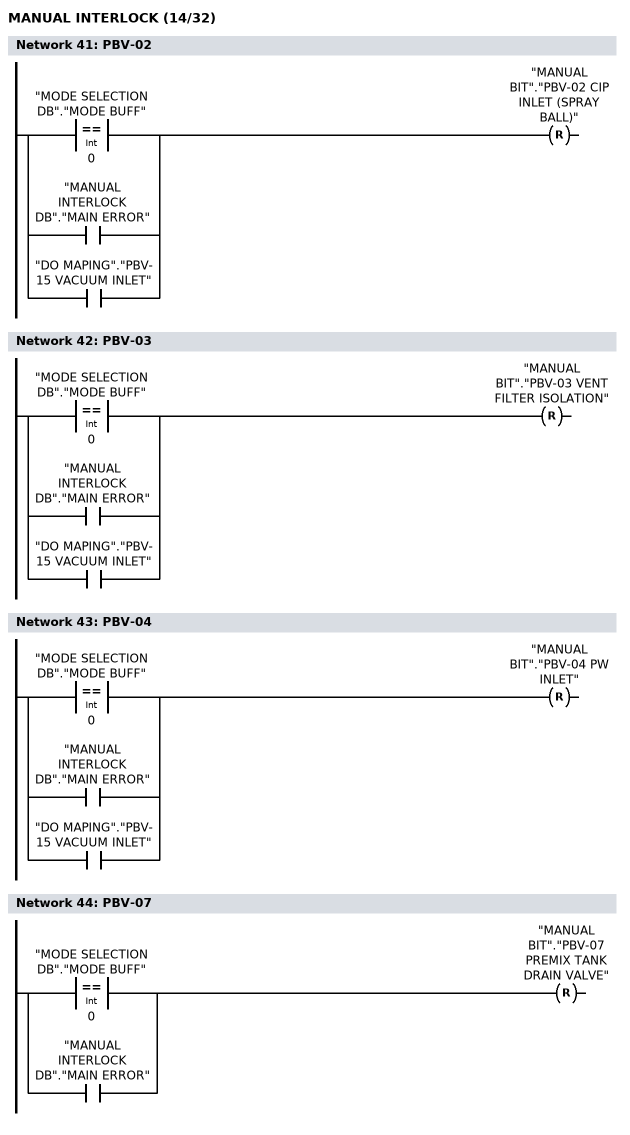
   RUNG wire#powerrail
      { S7_Templates := "SrcType := Int" } EQ_Contact(in1 := "MODE SELECTION DB"."MODE BUFF", in2 := 0)
      wire#w1
      R_Coil( "MANUAL BIT"."PBV-02 CIP INLET (SPRAY BALL)" )
   END_RUNG
   RUNG wire#powerrail
      Contact( "MANUAL INTERLOCK DB"."MAIN ERROR" )
   END_RUNG wire#w1
   RUNG wire#powerrail
      Contact( "DO MAPING"."PBV-15 VACUUM INLET" )
   END_RUNG wire#w1
   // the same network as SCL:
   IF ("MODE SELECTION DB"."MODE BUFF" = 0) OR "MANUAL INTERLOCK DB"."MAIN ERROR" OR "DO MAPING"."PBV-15 VACUUM INLET" THEN
       "MANUAL BIT"."PBV-02 CIP INLET (SPRAY BALL)" := FALSE;
   END_IF;
END_REGION

REGION Network 42: PBV-03
   RUNG wire#powerrail
      { S7_Templates := "SrcType := Int" } EQ_Contact(in1 := "MODE SELECTION DB"."MODE BUFF", in2 := 0)
      wire#w1
      R_Coil( "MANUAL BIT"."PBV-03 VENT FILTER ISOLATION" )
   END_RUNG
   RUNG wire#powerrail
      Contact( "MANUAL INTERLOCK DB"."MAIN ERROR" )
   END_RUNG wire#w1
   RUNG wire#powerrail
      Contact( "DO MAPING"."PBV-15 VACUUM INLET" )
   END_RUNG wire#w1
   // the same network as SCL:
   IF ("MODE SELECTION DB"."MODE BUFF" = 0) OR "MANUAL INTERLOCK DB"."MAIN ERROR" OR "DO MAPING"."PBV-15 VACUUM INLET" THEN
       "MANUAL BIT"."PBV-03 VENT FILTER ISOLATION" := FALSE;
   END_IF;
END_REGION

REGION Network 43: PBV-04
   RUNG wire#powerrail
      { S7_Templates := "SrcType := Int" } EQ_Contact(in1 := "MODE SELECTION DB"."MODE BUFF", in2 := 0)
      wire#w1
      R_Coil( "MANUAL BIT"."PBV-04 PW INLET" )
   END_RUNG
   RUNG wire#powerrail
      Contact( "MANUAL INTERLOCK DB"."MAIN ERROR" )
   END_RUNG wire#w1
   RUNG wire#powerrail
      Contact( "DO MAPING"."PBV-15 VACUUM INLET" )
   END_RUNG wire#w1
   // the same network as SCL:
   IF ("MODE SELECTION DB"."MODE BUFF" = 0) OR "MANUAL INTERLOCK DB"."MAIN ERROR" OR "DO MAPING"."PBV-15 VACUUM INLET" THEN
       "MANUAL BIT"."PBV-04 PW INLET" := FALSE;
   END_IF;
END_REGION

REGION Network 44: PBV-07
   RUNG wire#powerrail
      { S7_Templates := "SrcType := Int" } EQ_Contact(in1 := "MODE SELECTION DB"."MODE BUFF", in2 := 0)
      wire#w1
      R_Coil( "MANUAL BIT"."PBV-07 PREMIX TANK DRAIN VALVE" )
   END_RUNG
   RUNG wire#powerrail
      Contact( "MANUAL INTERLOCK DB"."MAIN ERROR" )
   END_RUNG wire#w1
   // the same network as SCL:
   IF ("MODE SELECTION DB"."MODE BUFF" = 0) OR "MANUAL INTERLOCK DB"."MAIN ERROR" THEN
       "MANUAL BIT"."PBV-07 PREMIX TANK DRAIN VALVE" := FALSE;
   END_IF;
END_REGION

REGION Network 45: PAV-09
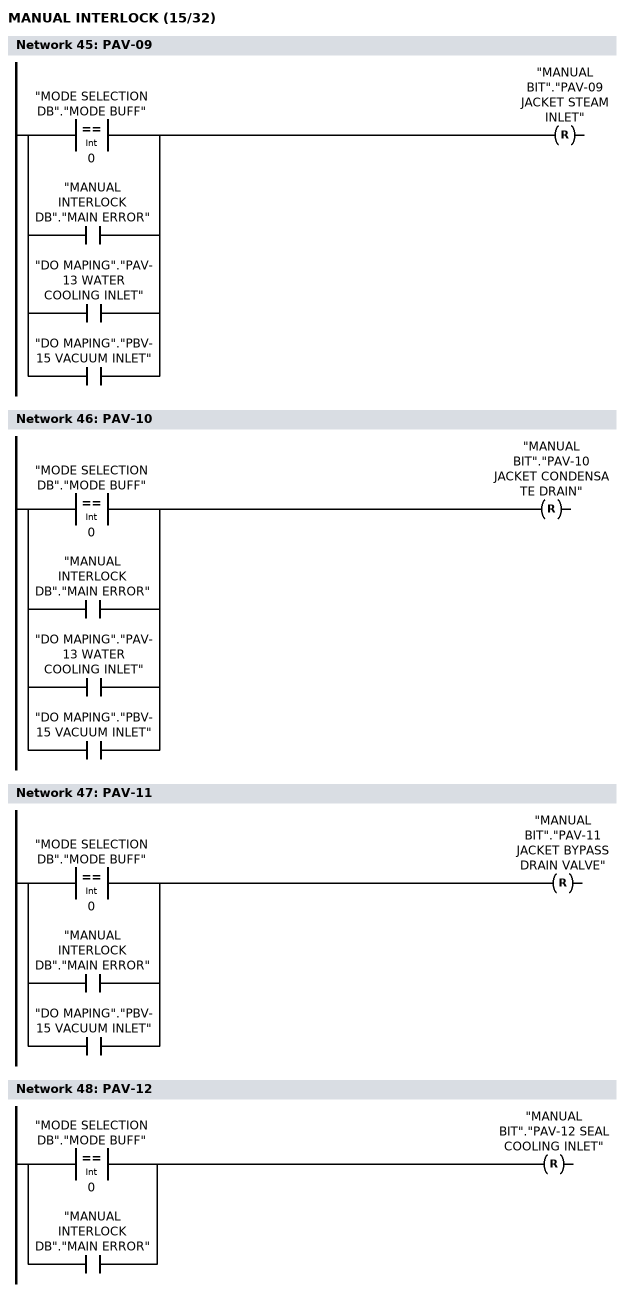
   RUNG wire#powerrail
      { S7_Templates := "SrcType := Int" } EQ_Contact(in1 := "MODE SELECTION DB"."MODE BUFF", in2 := 0)
      wire#w1
      R_Coil( "MANUAL BIT"."PAV-09 JACKET STEAM INLET" )
   END_RUNG
   RUNG wire#powerrail
      Contact( "MANUAL INTERLOCK DB"."MAIN ERROR" )
   END_RUNG wire#w1
   RUNG wire#powerrail
      Contact( "DO MAPING"."PAV-13 WATER COOLING INLET" )
   END_RUNG wire#w1
   RUNG wire#powerrail
      Contact( "DO MAPING"."PBV-15 VACUUM INLET" )
   END_RUNG wire#w1
   // the same network as SCL:
   IF ("MODE SELECTION DB"."MODE BUFF" = 0) OR "MANUAL INTERLOCK DB"."MAIN ERROR" OR "DO MAPING"."PAV-13 WATER COOLING INLET" OR "DO MAPING"."PBV-15 VACUUM INLET" THEN
       "MANUAL BIT"."PAV-09 JACKET STEAM INLET" := FALSE;
   END_IF;
END_REGION

REGION Network 46: PAV-10
   RUNG wire#powerrail
      { S7_Templates := "SrcType := Int" } EQ_Contact(in1 := "MODE SELECTION DB"."MODE BUFF", in2 := 0)
      wire#w1
      R_Coil( "MANUAL BIT"."PAV-10 JACKET CONDENSATE DRAIN" )
   END_RUNG
   RUNG wire#powerrail
      Contact( "MANUAL INTERLOCK DB"."MAIN ERROR" )
   END_RUNG wire#w1
   RUNG wire#powerrail
      Contact( "DO MAPING"."PAV-13 WATER COOLING INLET" )
   END_RUNG wire#w1
   RUNG wire#powerrail
      Contact( "DO MAPING"."PBV-15 VACUUM INLET" )
   END_RUNG wire#w1
   // the same network as SCL:
   IF ("MODE SELECTION DB"."MODE BUFF" = 0) OR "MANUAL INTERLOCK DB"."MAIN ERROR" OR "DO MAPING"."PAV-13 WATER COOLING INLET" OR "DO MAPING"."PBV-15 VACUUM INLET" THEN
       "MANUAL BIT"."PAV-10 JACKET CONDENSATE DRAIN" := FALSE;
   END_IF;
END_REGION

REGION Network 47: PAV-11
   RUNG wire#powerrail
      { S7_Templates := "SrcType := Int" } EQ_Contact(in1 := "MODE SELECTION DB"."MODE BUFF", in2 := 0)
      wire#w1
      R_Coil( "MANUAL BIT"."PAV-11 JACKET BYPASS DRAIN VALVE" )
   END_RUNG
   RUNG wire#powerrail
      Contact( "MANUAL INTERLOCK DB"."MAIN ERROR" )
   END_RUNG wire#w1
   RUNG wire#powerrail
      Contact( "DO MAPING"."PBV-15 VACUUM INLET" )
   END_RUNG wire#w1
   // the same network as SCL:
   IF ("MODE SELECTION DB"."MODE BUFF" = 0) OR "MANUAL INTERLOCK DB"."MAIN ERROR" OR "DO MAPING"."PBV-15 VACUUM INLET" THEN
       "MANUAL BIT"."PAV-11 JACKET BYPASS DRAIN VALVE" := FALSE;
   END_IF;
END_REGION

REGION Network 48: PAV-12
   RUNG wire#powerrail
      { S7_Templates := "SrcType := Int" } EQ_Contact(in1 := "MODE SELECTION DB"."MODE BUFF", in2 := 0)
      wire#w1
      R_Coil( "MANUAL BIT"."PAV-12 SEAL COOLING INLET" )
   END_RUNG
   RUNG wire#powerrail
      Contact( "MANUAL INTERLOCK DB"."MAIN ERROR" )
   END_RUNG wire#w1
   // the same network as SCL:
   IF ("MODE SELECTION DB"."MODE BUFF" = 0) OR "MANUAL INTERLOCK DB"."MAIN ERROR" THEN
       "MANUAL BIT"."PAV-12 SEAL COOLING INLET" := FALSE;
   END_IF;
END_REGION

REGION Network 49: PAV-13
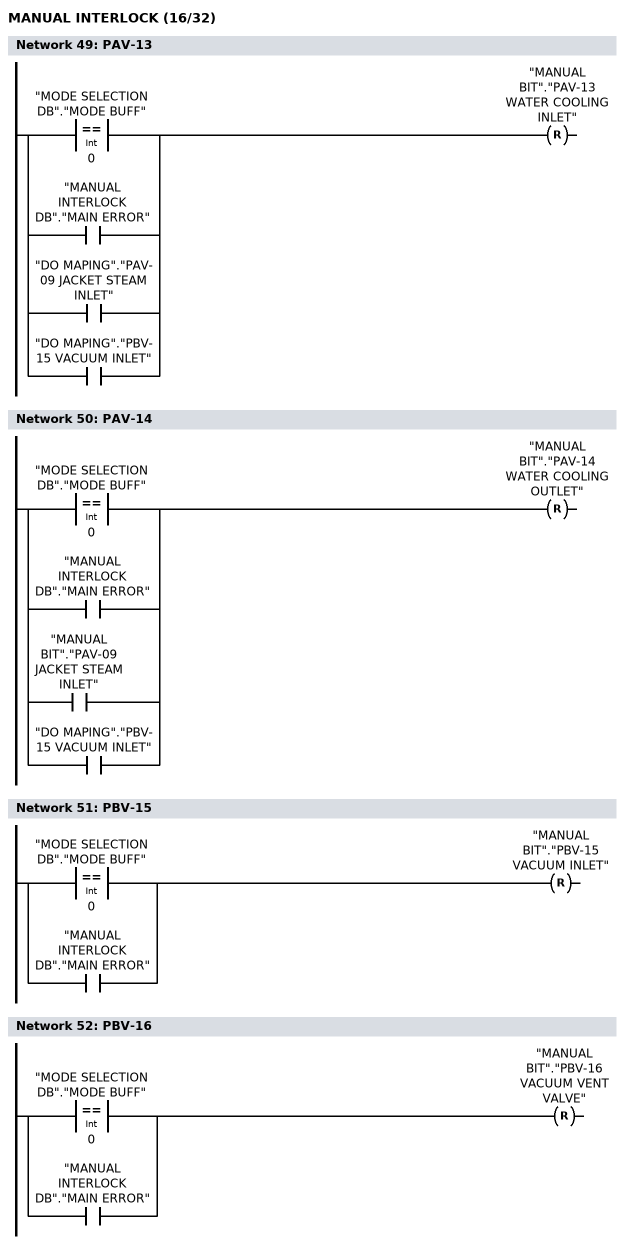
   RUNG wire#powerrail
      { S7_Templates := "SrcType := Int" } EQ_Contact(in1 := "MODE SELECTION DB"."MODE BUFF", in2 := 0)
      wire#w1
      R_Coil( "MANUAL BIT"."PAV-13 WATER COOLING INLET" )
   END_RUNG
   RUNG wire#powerrail
      Contact( "MANUAL INTERLOCK DB"."MAIN ERROR" )
   END_RUNG wire#w1
   RUNG wire#powerrail
      Contact( "DO MAPING"."PAV-09 JACKET STEAM INLET" )
   END_RUNG wire#w1
   RUNG wire#powerrail
      Contact( "DO MAPING"."PBV-15 VACUUM INLET" )
   END_RUNG wire#w1
   // the same network as SCL:
   IF ("MODE SELECTION DB"."MODE BUFF" = 0) OR "MANUAL INTERLOCK DB"."MAIN ERROR" OR "DO MAPING"."PAV-09 JACKET STEAM INLET" OR "DO MAPING"."PBV-15 VACUUM INLET" THEN
       "MANUAL BIT"."PAV-13 WATER COOLING INLET" := FALSE;
   END_IF;
END_REGION

REGION Network 50: PAV-14
   RUNG wire#powerrail
      { S7_Templates := "SrcType := Int" } EQ_Contact(in1 := "MODE SELECTION DB"."MODE BUFF", in2 := 0)
      wire#w1
      R_Coil( "MANUAL BIT"."PAV-14 WATER COOLING OUTLET" )
   END_RUNG
   RUNG wire#powerrail
      Contact( "MANUAL INTERLOCK DB"."MAIN ERROR" )
   END_RUNG wire#w1
   RUNG wire#powerrail
      Contact( "MANUAL BIT"."PAV-09 JACKET STEAM INLET" )
   END_RUNG wire#w1
   RUNG wire#powerrail
      Contact( "DO MAPING"."PBV-15 VACUUM INLET" )
   END_RUNG wire#w1
   // the same network as SCL:
   IF ("MODE SELECTION DB"."MODE BUFF" = 0) OR "MANUAL INTERLOCK DB"."MAIN ERROR" OR "MANUAL BIT"."PAV-09 JACKET STEAM INLET" OR "DO MAPING"."PBV-15 VACUUM INLET" THEN
       "MANUAL BIT"."PAV-14 WATER COOLING OUTLET" := FALSE;
   END_IF;
END_REGION

REGION Network 51: PBV-15
   RUNG wire#powerrail
      { S7_Templates := "SrcType := Int" } EQ_Contact(in1 := "MODE SELECTION DB"."MODE BUFF", in2 := 0)
      wire#w1
      R_Coil( "MANUAL BIT"."PBV-15 VACUUM INLET" )
   END_RUNG
   RUNG wire#powerrail
      Contact( "MANUAL INTERLOCK DB"."MAIN ERROR" )
   END_RUNG wire#w1
   // the same network as SCL:
   IF ("MODE SELECTION DB"."MODE BUFF" = 0) OR "MANUAL INTERLOCK DB"."MAIN ERROR" THEN
       "MANUAL BIT"."PBV-15 VACUUM INLET" := FALSE;
   END_IF;
END_REGION

REGION Network 52: PBV-16
   RUNG wire#powerrail
      { S7_Templates := "SrcType := Int" } EQ_Contact(in1 := "MODE SELECTION DB"."MODE BUFF", in2 := 0)
      wire#w1
      R_Coil( "MANUAL BIT"."PBV-16 VACUUM VENT VALVE" )
   END_RUNG
   RUNG wire#powerrail
      Contact( "MANUAL INTERLOCK DB"."MAIN ERROR" )
   END_RUNG wire#w1
   // the same network as SCL:
   IF ("MODE SELECTION DB"."MODE BUFF" = 0) OR "MANUAL INTERLOCK DB"."MAIN ERROR" THEN
       "MANUAL BIT"."PBV-16 VACUUM VENT VALVE" := FALSE;
   END_IF;
END_REGION

REGION Network 53: PFBV-17
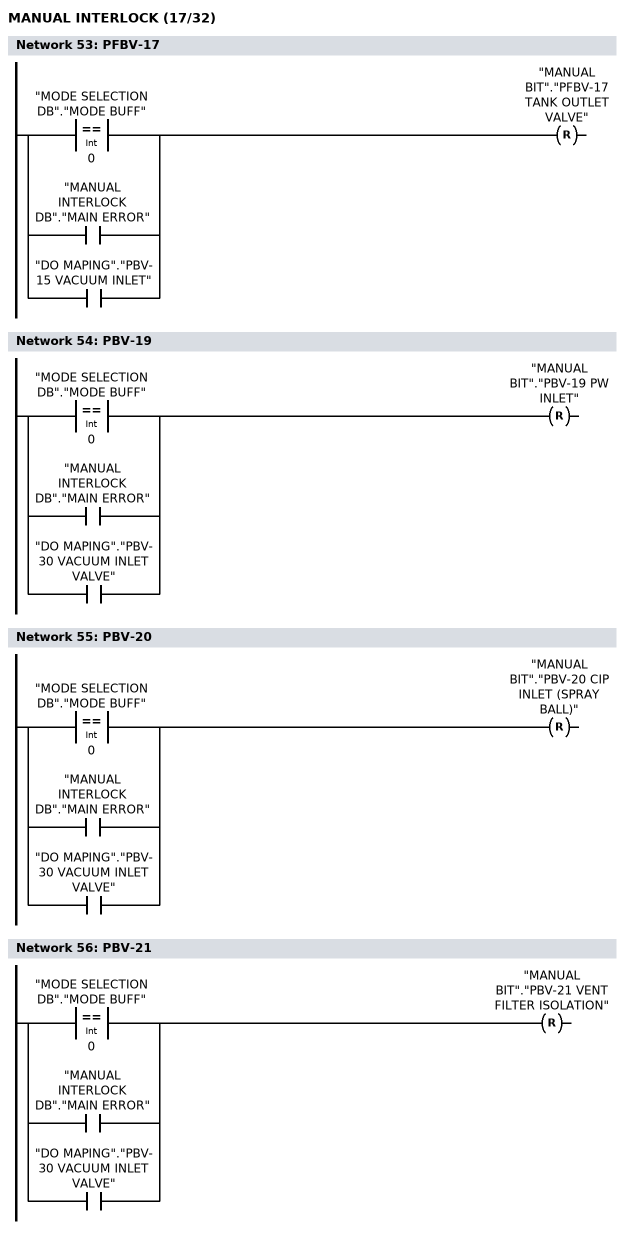
   RUNG wire#powerrail
      { S7_Templates := "SrcType := Int" } EQ_Contact(in1 := "MODE SELECTION DB"."MODE BUFF", in2 := 0)
      wire#w1
      R_Coil( "MANUAL BIT"."PFBV-17 TANK OUTLET VALVE" )
   END_RUNG
   RUNG wire#powerrail
      Contact( "MANUAL INTERLOCK DB"."MAIN ERROR" )
   END_RUNG wire#w1
   RUNG wire#powerrail
      Contact( "DO MAPING"."PBV-15 VACUUM INLET" )
   END_RUNG wire#w1
   // the same network as SCL:
   IF ("MODE SELECTION DB"."MODE BUFF" = 0) OR "MANUAL INTERLOCK DB"."MAIN ERROR" OR "DO MAPING"."PBV-15 VACUUM INLET" THEN
       "MANUAL BIT"."PFBV-17 TANK OUTLET VALVE" := FALSE;
   END_IF;
END_REGION

REGION Network 54: PBV-19
   RUNG wire#powerrail
      { S7_Templates := "SrcType := Int" } EQ_Contact(in1 := "MODE SELECTION DB"."MODE BUFF", in2 := 0)
      wire#w1
      R_Coil( "MANUAL BIT"."PBV-19 PW INLET" )
   END_RUNG
   RUNG wire#powerrail
      Contact( "MANUAL INTERLOCK DB"."MAIN ERROR" )
   END_RUNG wire#w1
   RUNG wire#powerrail
      Contact( "DO MAPING"."PBV-30 VACUUM INLET VALVE" )
   END_RUNG wire#w1
   // the same network as SCL:
   IF ("MODE SELECTION DB"."MODE BUFF" = 0) OR "MANUAL INTERLOCK DB"."MAIN ERROR" OR "DO MAPING"."PBV-30 VACUUM INLET VALVE" THEN
       "MANUAL BIT"."PBV-19 PW INLET" := FALSE;
   END_IF;
END_REGION

REGION Network 55: PBV-20
   RUNG wire#powerrail
      { S7_Templates := "SrcType := Int" } EQ_Contact(in1 := "MODE SELECTION DB"."MODE BUFF", in2 := 0)
      wire#w1
      R_Coil( "MANUAL BIT"."PBV-20 CIP INLET (SPRAY BALL)" )
   END_RUNG
   RUNG wire#powerrail
      Contact( "MANUAL INTERLOCK DB"."MAIN ERROR" )
   END_RUNG wire#w1
   RUNG wire#powerrail
      Contact( "DO MAPING"."PBV-30 VACUUM INLET VALVE" )
   END_RUNG wire#w1
   // the same network as SCL:
   IF ("MODE SELECTION DB"."MODE BUFF" = 0) OR "MANUAL INTERLOCK DB"."MAIN ERROR" OR "DO MAPING"."PBV-30 VACUUM INLET VALVE" THEN
       "MANUAL BIT"."PBV-20 CIP INLET (SPRAY BALL)" := FALSE;
   END_IF;
END_REGION

REGION Network 56: PBV-21
   RUNG wire#powerrail
      { S7_Templates := "SrcType := Int" } EQ_Contact(in1 := "MODE SELECTION DB"."MODE BUFF", in2 := 0)
      wire#w1
      R_Coil( "MANUAL BIT"."PBV-21 VENT FILTER ISOLATION" )
   END_RUNG
   RUNG wire#powerrail
      Contact( "MANUAL INTERLOCK DB"."MAIN ERROR" )
   END_RUNG wire#w1
   RUNG wire#powerrail
      Contact( "DO MAPING"."PBV-30 VACUUM INLET VALVE" )
   END_RUNG wire#w1
   // the same network as SCL:
   IF ("MODE SELECTION DB"."MODE BUFF" = 0) OR "MANUAL INTERLOCK DB"."MAIN ERROR" OR "DO MAPING"."PBV-30 VACUUM INLET VALVE" THEN
       "MANUAL BIT"."PBV-21 VENT FILTER ISOLATION" := FALSE;
   END_IF;
END_REGION

REGION Network 57: PBV-22
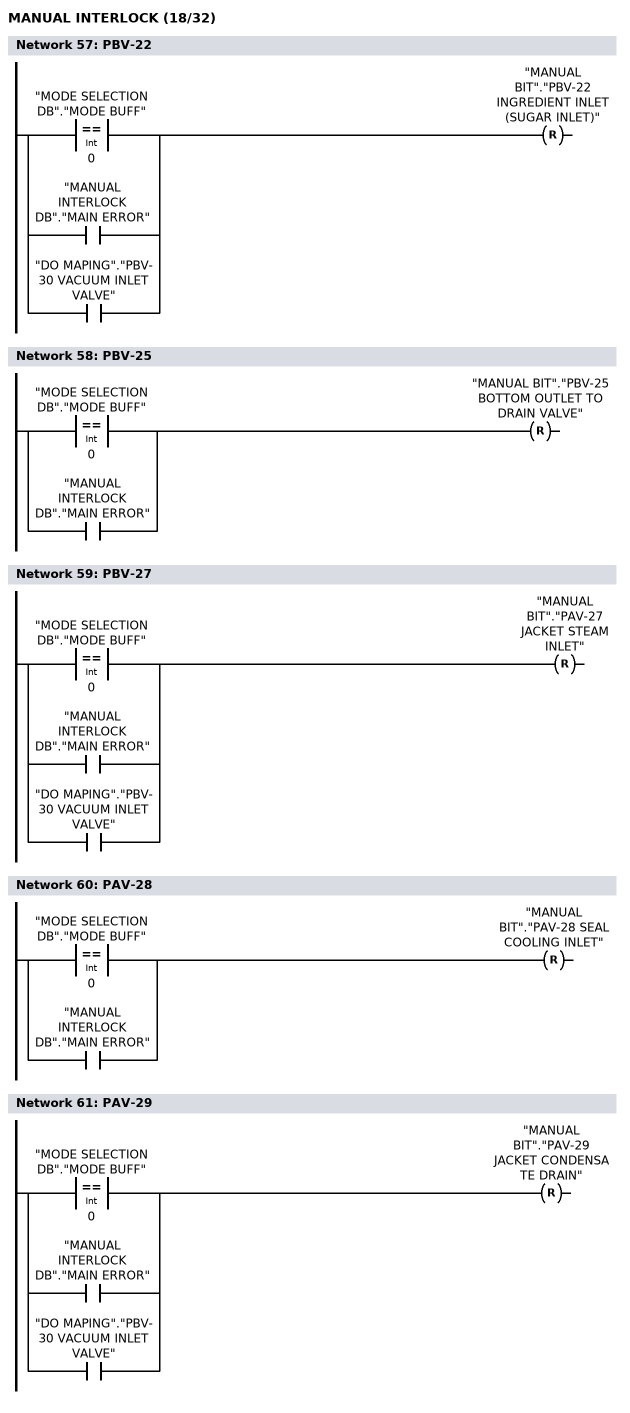
   RUNG wire#powerrail
      { S7_Templates := "SrcType := Int" } EQ_Contact(in1 := "MODE SELECTION DB"."MODE BUFF", in2 := 0)
      wire#w1
      R_Coil( "MANUAL BIT"."PBV-22 INGREDIENT INLET (SUGAR INLET)" )
   END_RUNG
   RUNG wire#powerrail
      Contact( "MANUAL INTERLOCK DB"."MAIN ERROR" )
   END_RUNG wire#w1
   RUNG wire#powerrail
      Contact( "DO MAPING"."PBV-30 VACUUM INLET VALVE" )
   END_RUNG wire#w1
   // the same network as SCL:
   IF ("MODE SELECTION DB"."MODE BUFF" = 0) OR "MANUAL INTERLOCK DB"."MAIN ERROR" OR "DO MAPING"."PBV-30 VACUUM INLET VALVE" THEN
       "MANUAL BIT"."PBV-22 INGREDIENT INLET (SUGAR INLET)" := FALSE;
   END_IF;
END_REGION

REGION Network 58: PBV-25
   RUNG wire#powerrail
      { S7_Templates := "SrcType := Int" } EQ_Contact(in1 := "MODE SELECTION DB"."MODE BUFF", in2 := 0)
      wire#w1
      R_Coil( "MANUAL BIT"."PBV-25 BOTTOM OUTLET TO DRAIN VALVE" )
   END_RUNG
   RUNG wire#powerrail
      Contact( "MANUAL INTERLOCK DB"."MAIN ERROR" )
   END_RUNG wire#w1
   // the same network as SCL:
   IF ("MODE SELECTION DB"."MODE BUFF" = 0) OR "MANUAL INTERLOCK DB"."MAIN ERROR" THEN
       "MANUAL BIT"."PBV-25 BOTTOM OUTLET TO DRAIN VALVE" := FALSE;
   END_IF;
END_REGION

REGION Network 59: PBV-27
   RUNG wire#powerrail
      { S7_Templates := "SrcType := Int" } EQ_Contact(in1 := "MODE SELECTION DB"."MODE BUFF", in2 := 0)
      wire#w1
      R_Coil( "MANUAL BIT"."PAV-27 JACKET STEAM INLET" )
   END_RUNG
   RUNG wire#powerrail
      Contact( "MANUAL INTERLOCK DB"."MAIN ERROR" )
   END_RUNG wire#w1
   RUNG wire#powerrail
      Contact( "DO MAPING"."PBV-30 VACUUM INLET VALVE" )
   END_RUNG wire#w1
   // the same network as SCL:
   IF ("MODE SELECTION DB"."MODE BUFF" = 0) OR "MANUAL INTERLOCK DB"."MAIN ERROR" OR "DO MAPING"."PBV-30 VACUUM INLET VALVE" THEN
       "MANUAL BIT"."PAV-27 JACKET STEAM INLET" := FALSE;
   END_IF;
END_REGION

REGION Network 60: PAV-28
   RUNG wire#powerrail
      { S7_Templates := "SrcType := Int" } EQ_Contact(in1 := "MODE SELECTION DB"."MODE BUFF", in2 := 0)
      wire#w1
      R_Coil( "MANUAL BIT"."PAV-28 SEAL COOLING INLET" )
   END_RUNG
   RUNG wire#powerrail
      Contact( "MANUAL INTERLOCK DB"."MAIN ERROR" )
   END_RUNG wire#w1
   // the same network as SCL:
   IF ("MODE SELECTION DB"."MODE BUFF" = 0) OR "MANUAL INTERLOCK DB"."MAIN ERROR" THEN
       "MANUAL BIT"."PAV-28 SEAL COOLING INLET" := FALSE;
   END_IF;
END_REGION

REGION Network 61: PAV-29
   RUNG wire#powerrail
      { S7_Templates := "SrcType := Int" } EQ_Contact(in1 := "MODE SELECTION DB"."MODE BUFF", in2 := 0)
      wire#w1
      R_Coil( "MANUAL BIT"."PAV-29 JACKET CONDENSATE DRAIN" )
   END_RUNG
   RUNG wire#powerrail
      Contact( "MANUAL INTERLOCK DB"."MAIN ERROR" )
   END_RUNG wire#w1
   RUNG wire#powerrail
      Contact( "DO MAPING"."PBV-30 VACUUM INLET VALVE" )
   END_RUNG wire#w1
   // the same network as SCL:
   IF ("MODE SELECTION DB"."MODE BUFF" = 0) OR "MANUAL INTERLOCK DB"."MAIN ERROR" OR "DO MAPING"."PBV-30 VACUUM INLET VALVE" THEN
       "MANUAL BIT"."PAV-29 JACKET CONDENSATE DRAIN" := FALSE;
   END_IF;
END_REGION

REGION Network 62: PBV-30
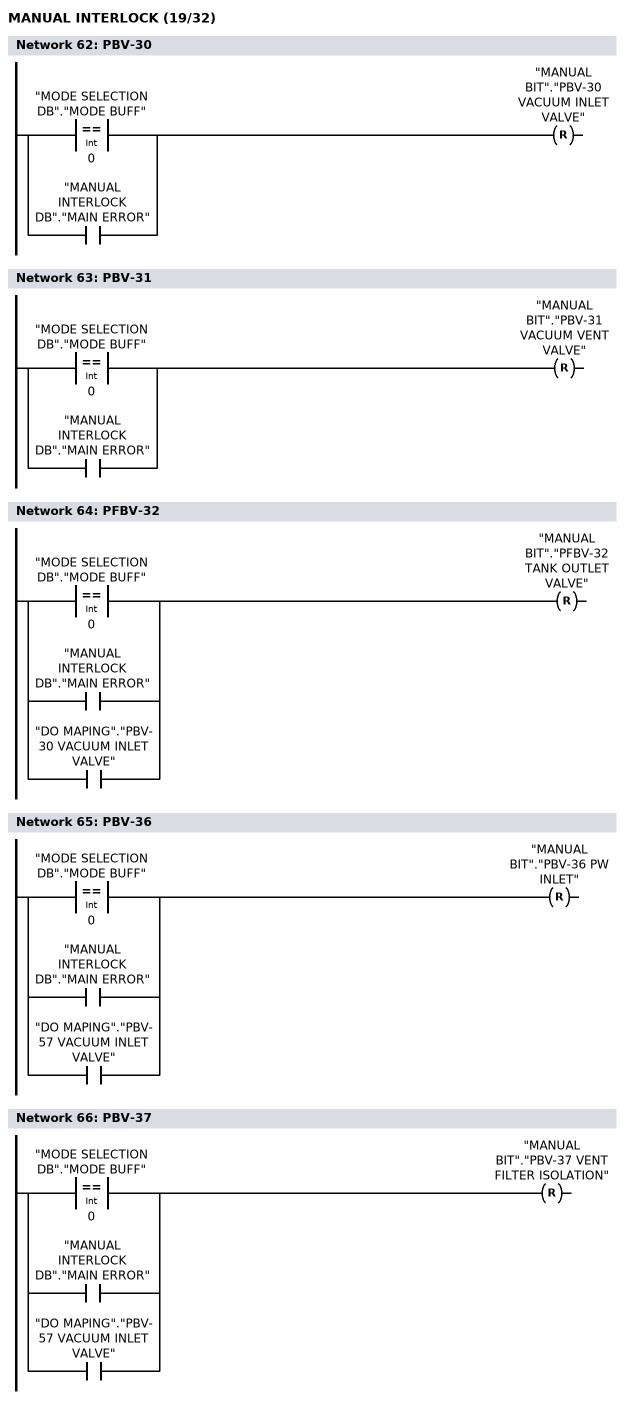
   RUNG wire#powerrail
      { S7_Templates := "SrcType := Int" } EQ_Contact(in1 := "MODE SELECTION DB"."MODE BUFF", in2 := 0)
      wire#w1
      R_Coil( "MANUAL BIT"."PBV-30 VACUUM INLET VALVE" )
   END_RUNG
   RUNG wire#powerrail
      Contact( "MANUAL INTERLOCK DB"."MAIN ERROR" )
   END_RUNG wire#w1
   // the same network as SCL:
   IF ("MODE SELECTION DB"."MODE BUFF" = 0) OR "MANUAL INTERLOCK DB"."MAIN ERROR" THEN
       "MANUAL BIT"."PBV-30 VACUUM INLET VALVE" := FALSE;
   END_IF;
END_REGION

REGION Network 63: PBV-31
   RUNG wire#powerrail
      { S7_Templates := "SrcType := Int" } EQ_Contact(in1 := "MODE SELECTION DB"."MODE BUFF", in2 := 0)
      wire#w1
      R_Coil( "MANUAL BIT"."PBV-31 VACUUM VENT VALVE" )
   END_RUNG
   RUNG wire#powerrail
      Contact( "MANUAL INTERLOCK DB"."MAIN ERROR" )
   END_RUNG wire#w1
   // the same network as SCL:
   IF ("MODE SELECTION DB"."MODE BUFF" = 0) OR "MANUAL INTERLOCK DB"."MAIN ERROR" THEN
       "MANUAL BIT"."PBV-31 VACUUM VENT VALVE" := FALSE;
   END_IF;
END_REGION

REGION Network 64: PFBV-32
   RUNG wire#powerrail
      { S7_Templates := "SrcType := Int" } EQ_Contact(in1 := "MODE SELECTION DB"."MODE BUFF", in2 := 0)
      wire#w1
      R_Coil( "MANUAL BIT"."PFBV-32 TANK OUTLET VALVE" )
   END_RUNG
   RUNG wire#powerrail
      Contact( "MANUAL INTERLOCK DB"."MAIN ERROR" )
   END_RUNG wire#w1
   RUNG wire#powerrail
      Contact( "DO MAPING"."PBV-30 VACUUM INLET VALVE" )
   END_RUNG wire#w1
   // the same network as SCL:
   IF ("MODE SELECTION DB"."MODE BUFF" = 0) OR "MANUAL INTERLOCK DB"."MAIN ERROR" OR "DO MAPING"."PBV-30 VACUUM INLET VALVE" THEN
       "MANUAL BIT"."PFBV-32 TANK OUTLET VALVE" := FALSE;
   END_IF;
END_REGION

REGION Network 65: PBV-36
   RUNG wire#powerrail
      { S7_Templates := "SrcType := Int" } EQ_Contact(in1 := "MODE SELECTION DB"."MODE BUFF", in2 := 0)
      wire#w1
      R_Coil( "MANUAL BIT"."PBV-36 PW INLET" )
   END_RUNG
   RUNG wire#powerrail
      Contact( "MANUAL INTERLOCK DB"."MAIN ERROR" )
   END_RUNG wire#w1
   RUNG wire#powerrail
      Contact( "DO MAPING"."PBV-57 VACUUM INLET VALVE" )
   END_RUNG wire#w1
   // the same network as SCL:
   IF ("MODE SELECTION DB"."MODE BUFF" = 0) OR "MANUAL INTERLOCK DB"."MAIN ERROR" OR "DO MAPING"."PBV-57 VACUUM INLET VALVE" THEN
       "MANUAL BIT"."PBV-36 PW INLET" := FALSE;
   END_IF;
END_REGION

REGION Network 66: PBV-37
   RUNG wire#powerrail
      { S7_Templates := "SrcType := Int" } EQ_Contact(in1 := "MODE SELECTION DB"."MODE BUFF", in2 := 0)
      wire#w1
      R_Coil( "MANUAL BIT"."PBV-37 VENT FILTER ISOLATION" )
   END_RUNG
   RUNG wire#powerrail
      Contact( "MANUAL INTERLOCK DB"."MAIN ERROR" )
   END_RUNG wire#w1
   RUNG wire#powerrail
      Contact( "DO MAPING"."PBV-57 VACUUM INLET VALVE" )
   END_RUNG wire#w1
   // the same network as SCL:
   IF ("MODE SELECTION DB"."MODE BUFF" = 0) OR "MANUAL INTERLOCK DB"."MAIN ERROR" OR "DO MAPING"."PBV-57 VACUUM INLET VALVE" THEN
       "MANUAL BIT"."PBV-37 VENT FILTER ISOLATION" := FALSE;
   END_IF;
END_REGION

REGION Network 67: PBV-38
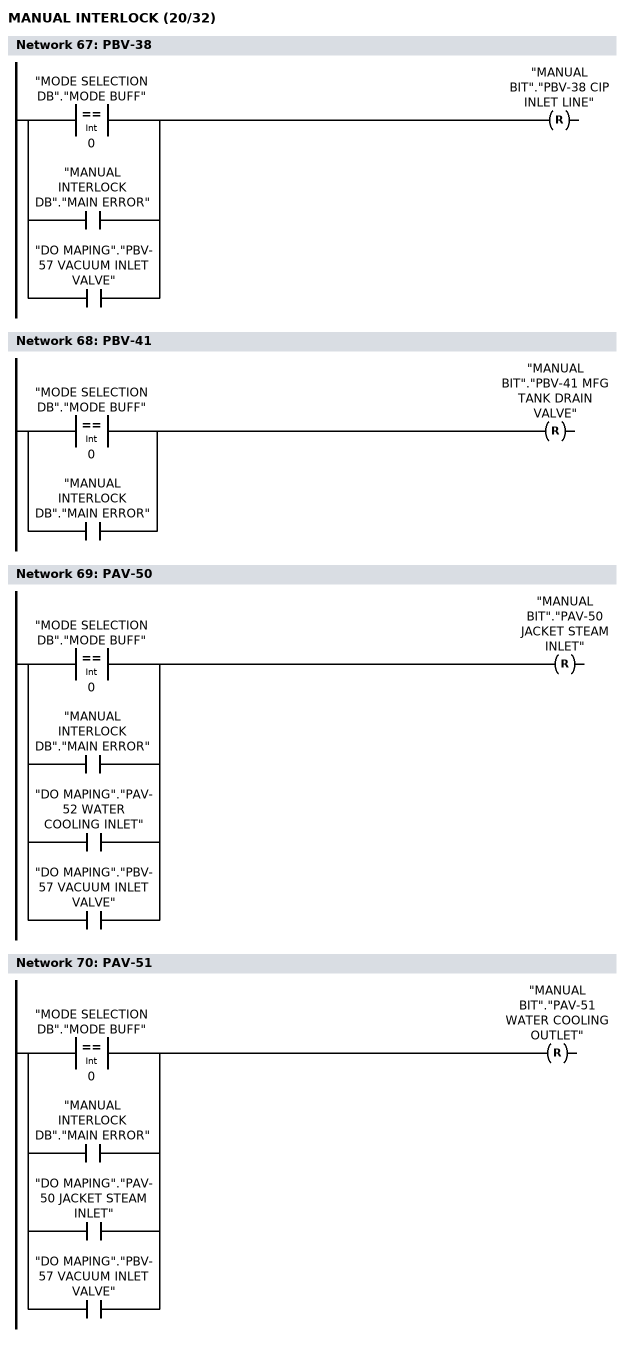
   RUNG wire#powerrail
      { S7_Templates := "SrcType := Int" } EQ_Contact(in1 := "MODE SELECTION DB"."MODE BUFF", in2 := 0)
      wire#w1
      R_Coil( "MANUAL BIT"."PBV-38 CIP INLET LINE" )
   END_RUNG
   RUNG wire#powerrail
      Contact( "MANUAL INTERLOCK DB"."MAIN ERROR" )
   END_RUNG wire#w1
   RUNG wire#powerrail
      Contact( "DO MAPING"."PBV-57 VACUUM INLET VALVE" )
   END_RUNG wire#w1
   // the same network as SCL:
   IF ("MODE SELECTION DB"."MODE BUFF" = 0) OR "MANUAL INTERLOCK DB"."MAIN ERROR" OR "DO MAPING"."PBV-57 VACUUM INLET VALVE" THEN
       "MANUAL BIT"."PBV-38 CIP INLET LINE" := FALSE;
   END_IF;
END_REGION

REGION Network 68: PBV-41
   RUNG wire#powerrail
      { S7_Templates := "SrcType := Int" } EQ_Contact(in1 := "MODE SELECTION DB"."MODE BUFF", in2 := 0)
      wire#w1
      R_Coil( "MANUAL BIT"."PBV-41 MFG TANK DRAIN VALVE" )
   END_RUNG
   RUNG wire#powerrail
      Contact( "MANUAL INTERLOCK DB"."MAIN ERROR" )
   END_RUNG wire#w1
   // the same network as SCL:
   IF ("MODE SELECTION DB"."MODE BUFF" = 0) OR "MANUAL INTERLOCK DB"."MAIN ERROR" THEN
       "MANUAL BIT"."PBV-41 MFG TANK DRAIN VALVE" := FALSE;
   END_IF;
END_REGION

REGION Network 69: PAV-50
   RUNG wire#powerrail
      { S7_Templates := "SrcType := Int" } EQ_Contact(in1 := "MODE SELECTION DB"."MODE BUFF", in2 := 0)
      wire#w1
      R_Coil( "MANUAL BIT"."PAV-50 JACKET STEAM INLET" )
   END_RUNG
   RUNG wire#powerrail
      Contact( "MANUAL INTERLOCK DB"."MAIN ERROR" )
   END_RUNG wire#w1
   RUNG wire#powerrail
      Contact( "DO MAPING"."PAV-52 WATER COOLING INLET" )
   END_RUNG wire#w1
   RUNG wire#powerrail
      Contact( "DO MAPING"."PBV-57 VACUUM INLET VALVE" )
   END_RUNG wire#w1
   // the same network as SCL:
   IF ("MODE SELECTION DB"."MODE BUFF" = 0) OR "MANUAL INTERLOCK DB"."MAIN ERROR" OR "DO MAPING"."PAV-52 WATER COOLING INLET" OR "DO MAPING"."PBV-57 VACUUM INLET VALVE" THEN
       "MANUAL BIT"."PAV-50 JACKET STEAM INLET" := FALSE;
   END_IF;
END_REGION

REGION Network 70: PAV-51
   RUNG wire#powerrail
      { S7_Templates := "SrcType := Int" } EQ_Contact(in1 := "MODE SELECTION DB"."MODE BUFF", in2 := 0)
      wire#w1
      R_Coil( "MANUAL BIT"."PAV-51 WATER COOLING OUTLET" )
   END_RUNG
   RUNG wire#powerrail
      Contact( "MANUAL INTERLOCK DB"."MAIN ERROR" )
   END_RUNG wire#w1
   RUNG wire#powerrail
      Contact( "DO MAPING"."PAV-50 JACKET STEAM INLET" )
   END_RUNG wire#w1
   RUNG wire#powerrail
      Contact( "DO MAPING"."PBV-57 VACUUM INLET VALVE" )
   END_RUNG wire#w1
   // the same network as SCL:
   IF ("MODE SELECTION DB"."MODE BUFF" = 0) OR "MANUAL INTERLOCK DB"."MAIN ERROR" OR "DO MAPING"."PAV-50 JACKET STEAM INLET" OR "DO MAPING"."PBV-57 VACUUM INLET VALVE" THEN
       "MANUAL BIT"."PAV-51 WATER COOLING OUTLET" := FALSE;
   END_IF;
END_REGION

REGION Network 71: PAV-52
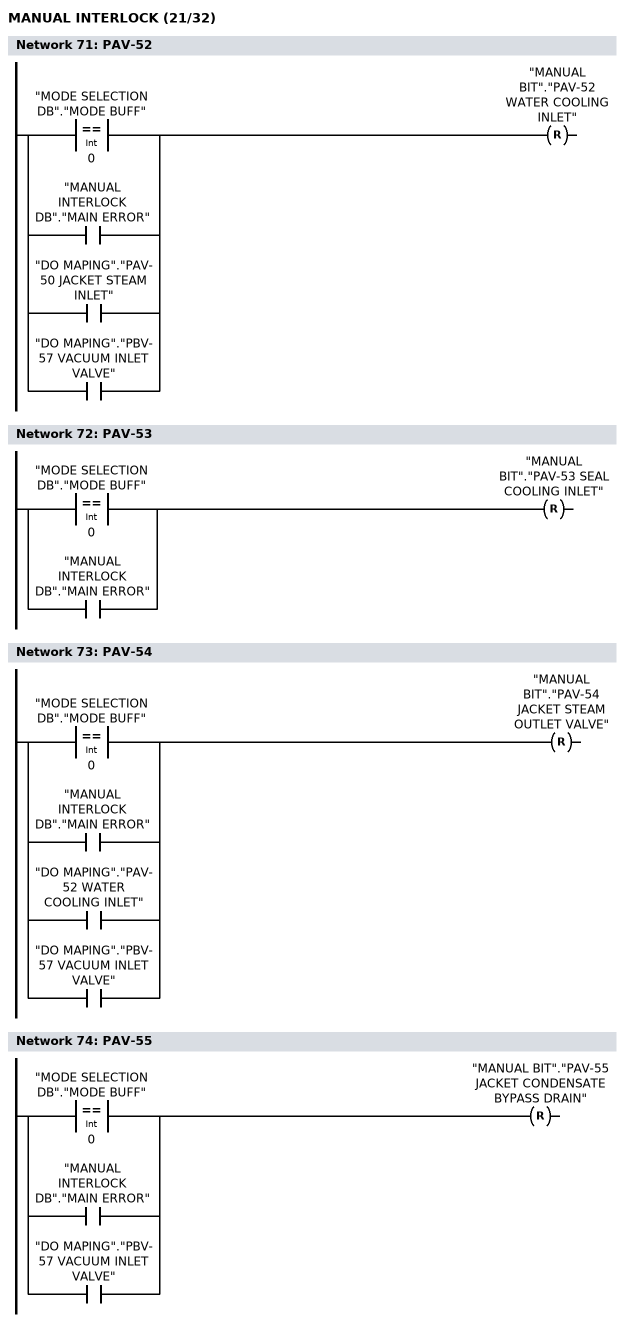
   RUNG wire#powerrail
      { S7_Templates := "SrcType := Int" } EQ_Contact(in1 := "MODE SELECTION DB"."MODE BUFF", in2 := 0)
      wire#w1
      R_Coil( "MANUAL BIT"."PAV-52 WATER COOLING INLET" )
   END_RUNG
   RUNG wire#powerrail
      Contact( "MANUAL INTERLOCK DB"."MAIN ERROR" )
   END_RUNG wire#w1
   RUNG wire#powerrail
      Contact( "DO MAPING"."PAV-50 JACKET STEAM INLET" )
   END_RUNG wire#w1
   RUNG wire#powerrail
      Contact( "DO MAPING"."PBV-57 VACUUM INLET VALVE" )
   END_RUNG wire#w1
   // the same network as SCL:
   IF ("MODE SELECTION DB"."MODE BUFF" = 0) OR "MANUAL INTERLOCK DB"."MAIN ERROR" OR "DO MAPING"."PAV-50 JACKET STEAM INLET" OR "DO MAPING"."PBV-57 VACUUM INLET VALVE" THEN
       "MANUAL BIT"."PAV-52 WATER COOLING INLET" := FALSE;
   END_IF;
END_REGION

REGION Network 72: PAV-53
   RUNG wire#powerrail
      { S7_Templates := "SrcType := Int" } EQ_Contact(in1 := "MODE SELECTION DB"."MODE BUFF", in2 := 0)
      wire#w1
      R_Coil( "MANUAL BIT"."PAV-53 SEAL COOLING INLET" )
   END_RUNG
   RUNG wire#powerrail
      Contact( "MANUAL INTERLOCK DB"."MAIN ERROR" )
   END_RUNG wire#w1
   // the same network as SCL:
   IF ("MODE SELECTION DB"."MODE BUFF" = 0) OR "MANUAL INTERLOCK DB"."MAIN ERROR" THEN
       "MANUAL BIT"."PAV-53 SEAL COOLING INLET" := FALSE;
   END_IF;
END_REGION

REGION Network 73: PAV-54
   RUNG wire#powerrail
      { S7_Templates := "SrcType := Int" } EQ_Contact(in1 := "MODE SELECTION DB"."MODE BUFF", in2 := 0)
      wire#w1
      R_Coil( "MANUAL BIT"."PAV-54 JACKET STEAM OUTLET VALVE" )
   END_RUNG
   RUNG wire#powerrail
      Contact( "MANUAL INTERLOCK DB"."MAIN ERROR" )
   END_RUNG wire#w1
   RUNG wire#powerrail
      Contact( "DO MAPING"."PAV-52 WATER COOLING INLET" )
   END_RUNG wire#w1
   RUNG wire#powerrail
      Contact( "DO MAPING"."PBV-57 VACUUM INLET VALVE" )
   END_RUNG wire#w1
   // the same network as SCL:
   IF ("MODE SELECTION DB"."MODE BUFF" = 0) OR "MANUAL INTERLOCK DB"."MAIN ERROR" OR "DO MAPING"."PAV-52 WATER COOLING INLET" OR "DO MAPING"."PBV-57 VACUUM INLET VALVE" THEN
       "MANUAL BIT"."PAV-54 JACKET STEAM OUTLET VALVE" := FALSE;
   END_IF;
END_REGION

REGION Network 74: PAV-55
   RUNG wire#powerrail
      { S7_Templates := "SrcType := Int" } EQ_Contact(in1 := "MODE SELECTION DB"."MODE BUFF", in2 := 0)
      wire#w1
      R_Coil( "MANUAL BIT"."PAV-55 JACKET CONDENSATE BYPASS DRAIN" )
   END_RUNG
   RUNG wire#powerrail
      Contact( "MANUAL INTERLOCK DB"."MAIN ERROR" )
   END_RUNG wire#w1
   RUNG wire#powerrail
      Contact( "DO MAPING"."PBV-57 VACUUM INLET VALVE" )
   END_RUNG wire#w1
   // the same network as SCL:
   IF ("MODE SELECTION DB"."MODE BUFF" = 0) OR "MANUAL INTERLOCK DB"."MAIN ERROR" OR "DO MAPING"."PBV-57 VACUUM INLET VALVE" THEN
       "MANUAL BIT"."PAV-55 JACKET CONDENSATE BYPASS DRAIN" := FALSE;
   END_IF;
END_REGION

REGION Network 75: PAV-56
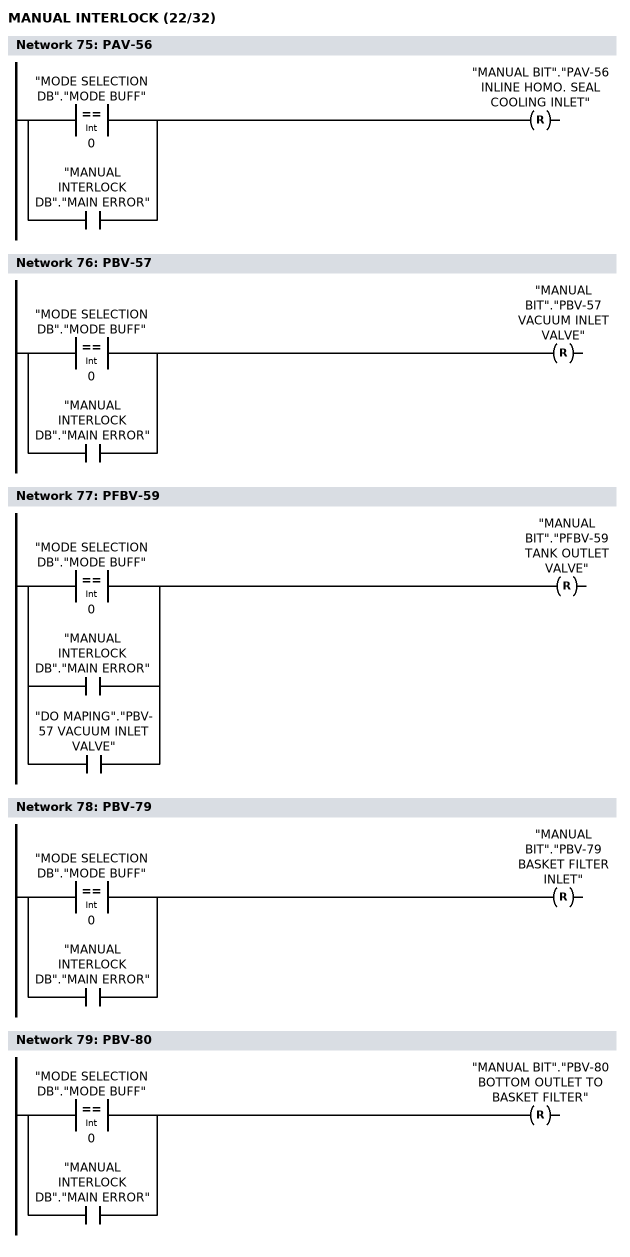
   RUNG wire#powerrail
      { S7_Templates := "SrcType := Int" } EQ_Contact(in1 := "MODE SELECTION DB"."MODE BUFF", in2 := 0)
      wire#w1
      R_Coil( "MANUAL BIT"."PAV-56 INLINE HOMO. SEAL COOLING INLET" )
   END_RUNG
   RUNG wire#powerrail
      Contact( "MANUAL INTERLOCK DB"."MAIN ERROR" )
   END_RUNG wire#w1
   // the same network as SCL:
   IF ("MODE SELECTION DB"."MODE BUFF" = 0) OR "MANUAL INTERLOCK DB"."MAIN ERROR" THEN
       "MANUAL BIT"."PAV-56 INLINE HOMO. SEAL COOLING INLET" := FALSE;
   END_IF;
END_REGION

REGION Network 76: PBV-57
   RUNG wire#powerrail
      { S7_Templates := "SrcType := Int" } EQ_Contact(in1 := "MODE SELECTION DB"."MODE BUFF", in2 := 0)
      wire#w1
      R_Coil( "MANUAL BIT"."PBV-57 VACUUM INLET VALVE" )
   END_RUNG
   RUNG wire#powerrail
      Contact( "MANUAL INTERLOCK DB"."MAIN ERROR" )
   END_RUNG wire#w1
   // the same network as SCL:
   IF ("MODE SELECTION DB"."MODE BUFF" = 0) OR "MANUAL INTERLOCK DB"."MAIN ERROR" THEN
       "MANUAL BIT"."PBV-57 VACUUM INLET VALVE" := FALSE;
   END_IF;
END_REGION

REGION Network 77: PFBV-59
   RUNG wire#powerrail
      { S7_Templates := "SrcType := Int" } EQ_Contact(in1 := "MODE SELECTION DB"."MODE BUFF", in2 := 0)
      wire#w1
      R_Coil( "MANUAL BIT"."PFBV-59 TANK OUTLET VALVE" )
   END_RUNG
   RUNG wire#powerrail
      Contact( "MANUAL INTERLOCK DB"."MAIN ERROR" )
   END_RUNG wire#w1
   RUNG wire#powerrail
      Contact( "DO MAPING"."PBV-57 VACUUM INLET VALVE" )
   END_RUNG wire#w1
   // the same network as SCL:
   IF ("MODE SELECTION DB"."MODE BUFF" = 0) OR "MANUAL INTERLOCK DB"."MAIN ERROR" OR "DO MAPING"."PBV-57 VACUUM INLET VALVE" THEN
       "MANUAL BIT"."PFBV-59 TANK OUTLET VALVE" := FALSE;
   END_IF;
END_REGION

REGION Network 78: PBV-79
   RUNG wire#powerrail
      { S7_Templates := "SrcType := Int" } EQ_Contact(in1 := "MODE SELECTION DB"."MODE BUFF", in2 := 0)
      wire#w1
      R_Coil( "MANUAL BIT"."PBV-79 BASKET FILTER INLET" )
   END_RUNG
   RUNG wire#powerrail
      Contact( "MANUAL INTERLOCK DB"."MAIN ERROR" )
   END_RUNG wire#w1
   // the same network as SCL:
   IF ("MODE SELECTION DB"."MODE BUFF" = 0) OR "MANUAL INTERLOCK DB"."MAIN ERROR" THEN
       "MANUAL BIT"."PBV-79 BASKET FILTER INLET" := FALSE;
   END_IF;
END_REGION

REGION Network 79: PBV-80
   RUNG wire#powerrail
      { S7_Templates := "SrcType := Int" } EQ_Contact(in1 := "MODE SELECTION DB"."MODE BUFF", in2 := 0)
      wire#w1
      R_Coil( "MANUAL BIT"."PBV-80 BOTTOM OUTLET TO BASKET FILTER" )
   END_RUNG
   RUNG wire#powerrail
      Contact( "MANUAL INTERLOCK DB"."MAIN ERROR" )
   END_RUNG wire#w1
   // the same network as SCL:
   IF ("MODE SELECTION DB"."MODE BUFF" = 0) OR "MANUAL INTERLOCK DB"."MAIN ERROR" THEN
       "MANUAL BIT"."PBV-80 BOTTOM OUTLET TO BASKET FILTER" := FALSE;
   END_IF;
END_REGION

REGION Network 80: PBV-81
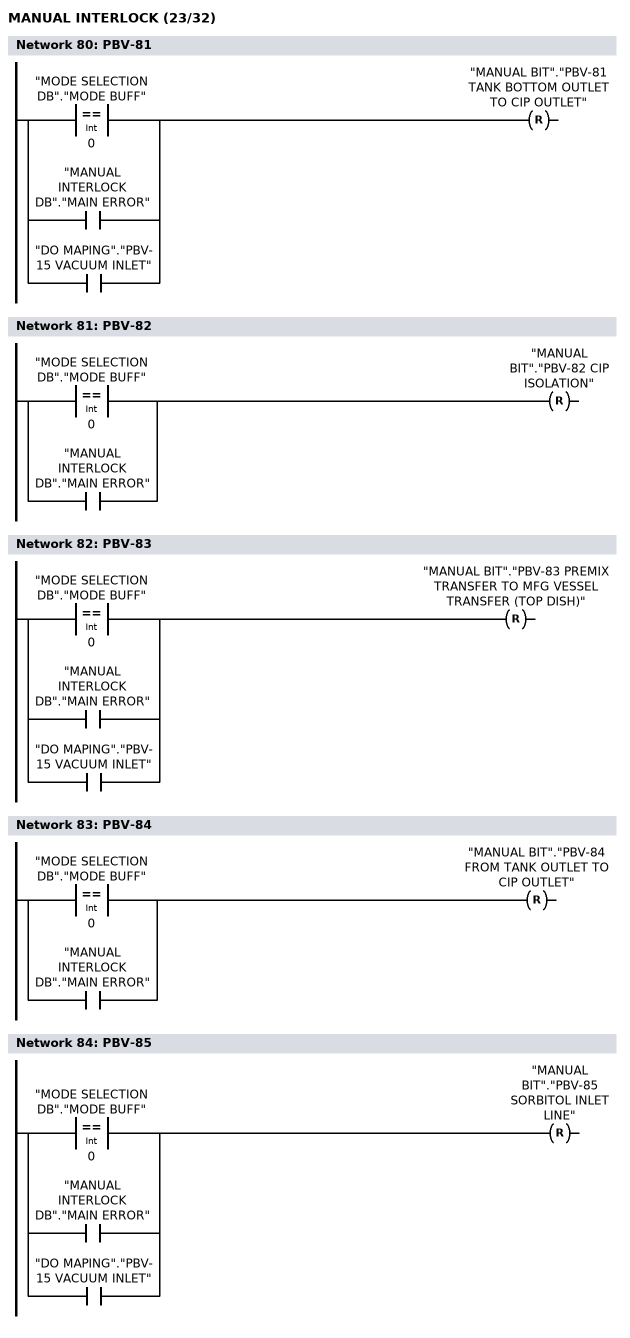
   RUNG wire#powerrail
      { S7_Templates := "SrcType := Int" } EQ_Contact(in1 := "MODE SELECTION DB"."MODE BUFF", in2 := 0)
      wire#w1
      R_Coil( "MANUAL BIT"."PBV-81 TANK BOTTOM OUTLET TO CIP OUTLET" )
   END_RUNG
   RUNG wire#powerrail
      Contact( "MANUAL INTERLOCK DB"."MAIN ERROR" )
   END_RUNG wire#w1
   RUNG wire#powerrail
      Contact( "DO MAPING"."PBV-15 VACUUM INLET" )
   END_RUNG wire#w1
   // the same network as SCL:
   IF ("MODE SELECTION DB"."MODE BUFF" = 0) OR "MANUAL INTERLOCK DB"."MAIN ERROR" OR "DO MAPING"."PBV-15 VACUUM INLET" THEN
       "MANUAL BIT"."PBV-81 TANK BOTTOM OUTLET TO CIP OUTLET" := FALSE;
   END_IF;
END_REGION

REGION Network 81: PBV-82
   RUNG wire#powerrail
      { S7_Templates := "SrcType := Int" } EQ_Contact(in1 := "MODE SELECTION DB"."MODE BUFF", in2 := 0)
      wire#w1
      R_Coil( "MANUAL BIT"."PBV-82 CIP ISOLATION" )
   END_RUNG
   RUNG wire#powerrail
      Contact( "MANUAL INTERLOCK DB"."MAIN ERROR" )
   END_RUNG wire#w1
   // the same network as SCL:
   IF ("MODE SELECTION DB"."MODE BUFF" = 0) OR "MANUAL INTERLOCK DB"."MAIN ERROR" THEN
       "MANUAL BIT"."PBV-82 CIP ISOLATION" := FALSE;
   END_IF;
END_REGION

REGION Network 82: PBV-83
   RUNG wire#powerrail
      { S7_Templates := "SrcType := Int" } EQ_Contact(in1 := "MODE SELECTION DB"."MODE BUFF", in2 := 0)
      wire#w1
      R_Coil( "MANUAL BIT"."PBV-83 PREMIX TRANSFER TO MFG VESSEL TRANSFER (TOP DISH)" )
   END_RUNG
   RUNG wire#powerrail
      Contact( "MANUAL INTERLOCK DB"."MAIN ERROR" )
   END_RUNG wire#w1
   RUNG wire#powerrail
      Contact( "DO MAPING"."PBV-15 VACUUM INLET" )
   END_RUNG wire#w1
   // the same network as SCL:
   IF ("MODE SELECTION DB"."MODE BUFF" = 0) OR "MANUAL INTERLOCK DB"."MAIN ERROR" OR "DO MAPING"."PBV-15 VACUUM INLET" THEN
       "MANUAL BIT"."PBV-83 PREMIX TRANSFER TO MFG VESSEL TRANSFER (TOP DISH)" := FALSE;
   END_IF;
END_REGION

REGION Network 83: PBV-84
   RUNG wire#powerrail
      { S7_Templates := "SrcType := Int" } EQ_Contact(in1 := "MODE SELECTION DB"."MODE BUFF", in2 := 0)
      wire#w1
      R_Coil( "MANUAL BIT"."PBV-84 FROM TANK OUTLET TO CIP OUTLET" )
   END_RUNG
   RUNG wire#powerrail
      Contact( "MANUAL INTERLOCK DB"."MAIN ERROR" )
   END_RUNG wire#w1
   // the same network as SCL:
   IF ("MODE SELECTION DB"."MODE BUFF" = 0) OR "MANUAL INTERLOCK DB"."MAIN ERROR" THEN
       "MANUAL BIT"."PBV-84 FROM TANK OUTLET TO CIP OUTLET" := FALSE;
   END_IF;
END_REGION

REGION Network 84: PBV-85
   RUNG wire#powerrail
      { S7_Templates := "SrcType := Int" } EQ_Contact(in1 := "MODE SELECTION DB"."MODE BUFF", in2 := 0)
      wire#w1
      R_Coil( "MANUAL BIT"."PBV-85 SORBITOL INLET LINE" )
   END_RUNG
   RUNG wire#powerrail
      Contact( "MANUAL INTERLOCK DB"."MAIN ERROR" )
   END_RUNG wire#w1
   RUNG wire#powerrail
      Contact( "DO MAPING"."PBV-15 VACUUM INLET" )
   END_RUNG wire#w1
   // the same network as SCL:
   IF ("MODE SELECTION DB"."MODE BUFF" = 0) OR "MANUAL INTERLOCK DB"."MAIN ERROR" OR "DO MAPING"."PBV-15 VACUUM INLET" THEN
       "MANUAL BIT"."PBV-85 SORBITOL INLET LINE" := FALSE;
   END_IF;
END_REGION

REGION Network 85: PBV-86
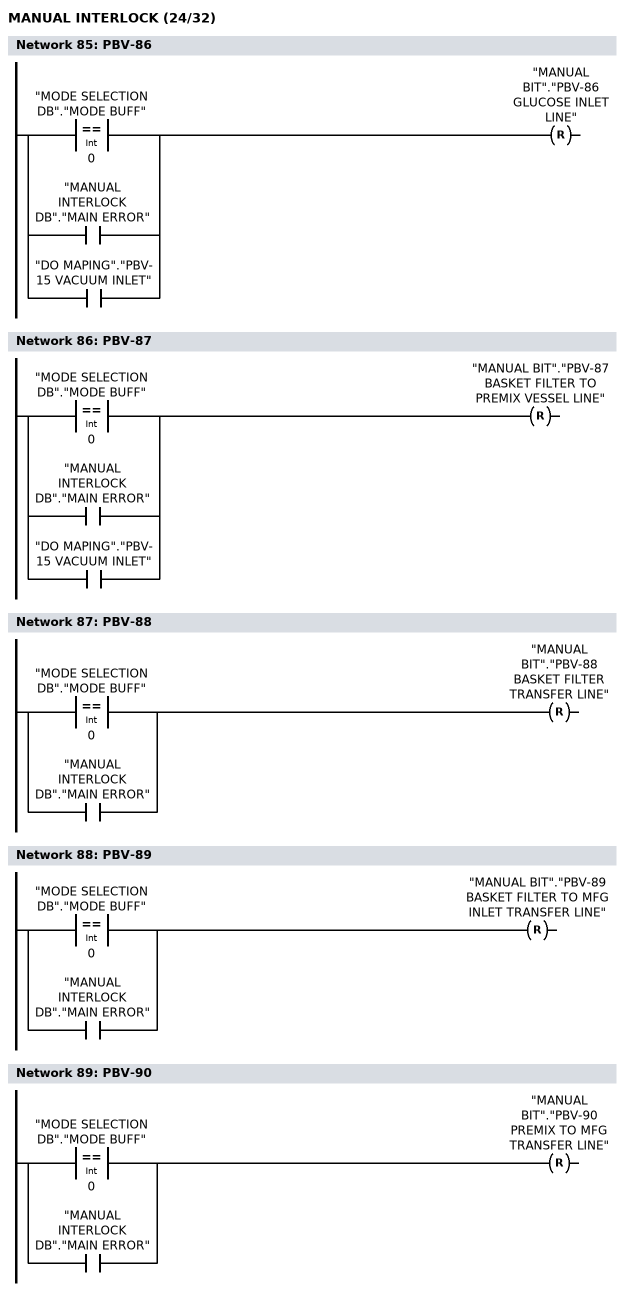
   RUNG wire#powerrail
      { S7_Templates := "SrcType := Int" } EQ_Contact(in1 := "MODE SELECTION DB"."MODE BUFF", in2 := 0)
      wire#w1
      R_Coil( "MANUAL BIT"."PBV-86 GLUCOSE INLET LINE" )
   END_RUNG
   RUNG wire#powerrail
      Contact( "MANUAL INTERLOCK DB"."MAIN ERROR" )
   END_RUNG wire#w1
   RUNG wire#powerrail
      Contact( "DO MAPING"."PBV-15 VACUUM INLET" )
   END_RUNG wire#w1
   // the same network as SCL:
   IF ("MODE SELECTION DB"."MODE BUFF" = 0) OR "MANUAL INTERLOCK DB"."MAIN ERROR" OR "DO MAPING"."PBV-15 VACUUM INLET" THEN
       "MANUAL BIT"."PBV-86 GLUCOSE INLET LINE" := FALSE;
   END_IF;
END_REGION

REGION Network 86: PBV-87
   RUNG wire#powerrail
      { S7_Templates := "SrcType := Int" } EQ_Contact(in1 := "MODE SELECTION DB"."MODE BUFF", in2 := 0)
      wire#w1
      R_Coil( "MANUAL BIT"."PBV-87 BASKET FILTER TO PREMIX VESSEL LINE" )
   END_RUNG
   RUNG wire#powerrail
      Contact( "MANUAL INTERLOCK DB"."MAIN ERROR" )
   END_RUNG wire#w1
   RUNG wire#powerrail
      Contact( "DO MAPING"."PBV-15 VACUUM INLET" )
   END_RUNG wire#w1
   // the same network as SCL:
   IF ("MODE SELECTION DB"."MODE BUFF" = 0) OR "MANUAL INTERLOCK DB"."MAIN ERROR" OR "DO MAPING"."PBV-15 VACUUM INLET" THEN
       "MANUAL BIT"."PBV-87 BASKET FILTER TO PREMIX VESSEL LINE" := FALSE;
   END_IF;
END_REGION

REGION Network 87: PBV-88
   RUNG wire#powerrail
      { S7_Templates := "SrcType := Int" } EQ_Contact(in1 := "MODE SELECTION DB"."MODE BUFF", in2 := 0)
      wire#w1
      R_Coil( "MANUAL BIT"."PBV-88 BASKET FILTER TRANSFER LINE" )
   END_RUNG
   RUNG wire#powerrail
      Contact( "MANUAL INTERLOCK DB"."MAIN ERROR" )
   END_RUNG wire#w1
   // the same network as SCL:
   IF ("MODE SELECTION DB"."MODE BUFF" = 0) OR "MANUAL INTERLOCK DB"."MAIN ERROR" THEN
       "MANUAL BIT"."PBV-88 BASKET FILTER TRANSFER LINE" := FALSE;
   END_IF;
END_REGION

REGION Network 88: PBV-89
   RUNG wire#powerrail
      { S7_Templates := "SrcType := Int" } EQ_Contact(in1 := "MODE SELECTION DB"."MODE BUFF", in2 := 0)
      wire#w1
      R_Coil( "MANUAL BIT"."PBV-89 BASKET FILTER TO MFG INLET TRANSFER LINE" )
   END_RUNG
   RUNG wire#powerrail
      Contact( "MANUAL INTERLOCK DB"."MAIN ERROR" )
   END_RUNG wire#w1
   // the same network as SCL:
   IF ("MODE SELECTION DB"."MODE BUFF" = 0) OR "MANUAL INTERLOCK DB"."MAIN ERROR" THEN
       "MANUAL BIT"."PBV-89 BASKET FILTER TO MFG INLET TRANSFER LINE" := FALSE;
   END_IF;
END_REGION

REGION Network 89: PBV-90
   RUNG wire#powerrail
      { S7_Templates := "SrcType := Int" } EQ_Contact(in1 := "MODE SELECTION DB"."MODE BUFF", in2 := 0)
      wire#w1
      R_Coil( "MANUAL BIT"."PBV-90 PREMIX TO MFG TRANSFER LINE" )
   END_RUNG
   RUNG wire#powerrail
      Contact( "MANUAL INTERLOCK DB"."MAIN ERROR" )
   END_RUNG wire#w1
   // the same network as SCL:
   IF ("MODE SELECTION DB"."MODE BUFF" = 0) OR "MANUAL INTERLOCK DB"."MAIN ERROR" THEN
       "MANUAL BIT"."PBV-90 PREMIX TO MFG TRANSFER LINE" := FALSE;
   END_IF;
END_REGION

REGION Network 90: PBV-91
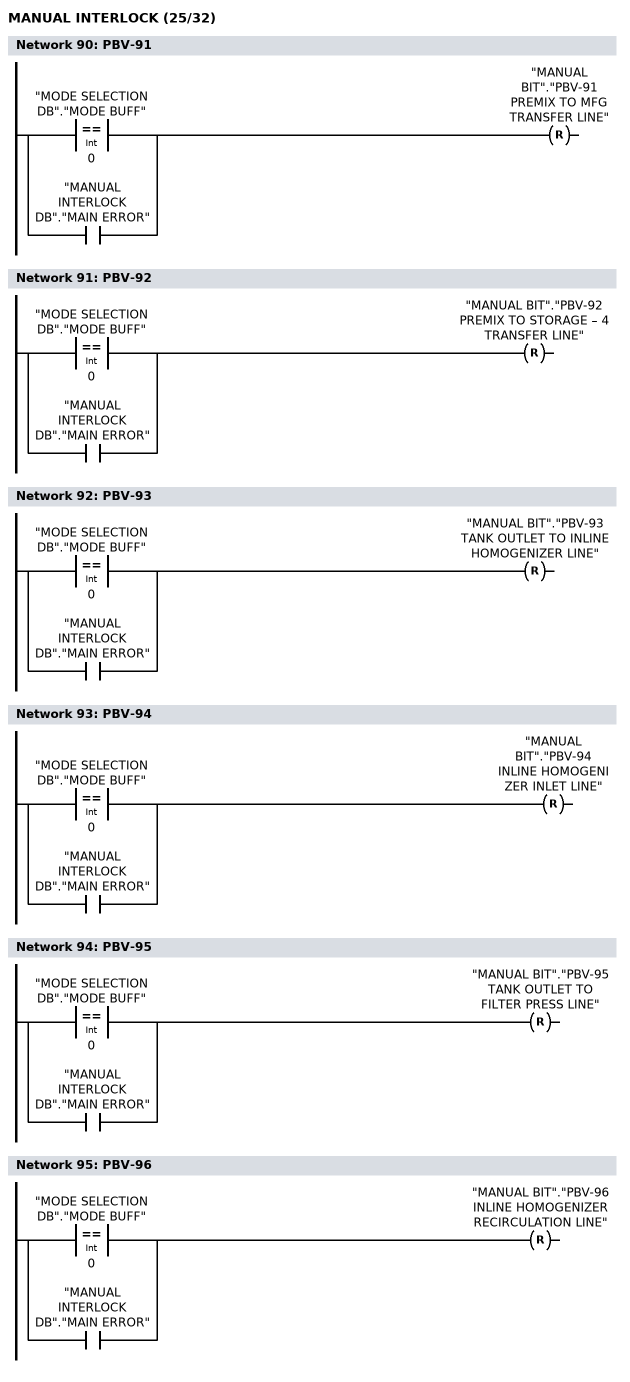
   RUNG wire#powerrail
      { S7_Templates := "SrcType := Int" } EQ_Contact(in1 := "MODE SELECTION DB"."MODE BUFF", in2 := 0)
      wire#w1
      R_Coil( "MANUAL BIT"."PBV-91 PREMIX TO MFG TRANSFER LINE" )
   END_RUNG
   RUNG wire#powerrail
      Contact( "MANUAL INTERLOCK DB"."MAIN ERROR" )
   END_RUNG wire#w1
   // the same network as SCL:
   IF ("MODE SELECTION DB"."MODE BUFF" = 0) OR "MANUAL INTERLOCK DB"."MAIN ERROR" THEN
       "MANUAL BIT"."PBV-91 PREMIX TO MFG TRANSFER LINE" := FALSE;
   END_IF;
END_REGION

REGION Network 91: PBV-92
   RUNG wire#powerrail
      { S7_Templates := "SrcType := Int" } EQ_Contact(in1 := "MODE SELECTION DB"."MODE BUFF", in2 := 0)
      wire#w1
      R_Coil( "MANUAL BIT"."PBV-92 PREMIX TO STORAGE – 4 TRANSFER LINE" )
   END_RUNG
   RUNG wire#powerrail
      Contact( "MANUAL INTERLOCK DB"."MAIN ERROR" )
   END_RUNG wire#w1
   // the same network as SCL:
   IF ("MODE SELECTION DB"."MODE BUFF" = 0) OR "MANUAL INTERLOCK DB"."MAIN ERROR" THEN
       "MANUAL BIT"."PBV-92 PREMIX TO STORAGE – 4 TRANSFER LINE" := FALSE;
   END_IF;
END_REGION

REGION Network 92: PBV-93
   RUNG wire#powerrail
      { S7_Templates := "SrcType := Int" } EQ_Contact(in1 := "MODE SELECTION DB"."MODE BUFF", in2 := 0)
      wire#w1
      R_Coil( "MANUAL BIT"."PBV-93 TANK OUTLET TO INLINE HOMOGENIZER LINE" )
   END_RUNG
   RUNG wire#powerrail
      Contact( "MANUAL INTERLOCK DB"."MAIN ERROR" )
   END_RUNG wire#w1
   // the same network as SCL:
   IF ("MODE SELECTION DB"."MODE BUFF" = 0) OR "MANUAL INTERLOCK DB"."MAIN ERROR" THEN
       "MANUAL BIT"."PBV-93 TANK OUTLET TO INLINE HOMOGENIZER LINE" := FALSE;
   END_IF;
END_REGION

REGION Network 93: PBV-94
   RUNG wire#powerrail
      { S7_Templates := "SrcType := Int" } EQ_Contact(in1 := "MODE SELECTION DB"."MODE BUFF", in2 := 0)
      wire#w1
      R_Coil( "MANUAL BIT"."PBV-94 INLINE HOMOGENIZER INLET LINE" )
   END_RUNG
   RUNG wire#powerrail
      Contact( "MANUAL INTERLOCK DB"."MAIN ERROR" )
   END_RUNG wire#w1
   // the same network as SCL:
   IF ("MODE SELECTION DB"."MODE BUFF" = 0) OR "MANUAL INTERLOCK DB"."MAIN ERROR" THEN
       "MANUAL BIT"."PBV-94 INLINE HOMOGENIZER INLET LINE" := FALSE;
   END_IF;
END_REGION

REGION Network 94: PBV-95
   RUNG wire#powerrail
      { S7_Templates := "SrcType := Int" } EQ_Contact(in1 := "MODE SELECTION DB"."MODE BUFF", in2 := 0)
      wire#w1
      R_Coil( "MANUAL BIT"."PBV-95 TANK OUTLET TO FILTER PRESS LINE" )
   END_RUNG
   RUNG wire#powerrail
      Contact( "MANUAL INTERLOCK DB"."MAIN ERROR" )
   END_RUNG wire#w1
   // the same network as SCL:
   IF ("MODE SELECTION DB"."MODE BUFF" = 0) OR "MANUAL INTERLOCK DB"."MAIN ERROR" THEN
       "MANUAL BIT"."PBV-95 TANK OUTLET TO FILTER PRESS LINE" := FALSE;
   END_IF;
END_REGION

REGION Network 95: PBV-96
   RUNG wire#powerrail
      { S7_Templates := "SrcType := Int" } EQ_Contact(in1 := "MODE SELECTION DB"."MODE BUFF", in2 := 0)
      wire#w1
      R_Coil( "MANUAL BIT"."PBV-96 INLINE HOMOGENIZER RECIRCULATION LINE" )
   END_RUNG
   RUNG wire#powerrail
      Contact( "MANUAL INTERLOCK DB"."MAIN ERROR" )
   END_RUNG wire#w1
   // the same network as SCL:
   IF ("MODE SELECTION DB"."MODE BUFF" = 0) OR "MANUAL INTERLOCK DB"."MAIN ERROR" THEN
       "MANUAL BIT"."PBV-96 INLINE HOMOGENIZER RECIRCULATION LINE" := FALSE;
   END_IF;
END_REGION

REGION Network 96: PBV-97
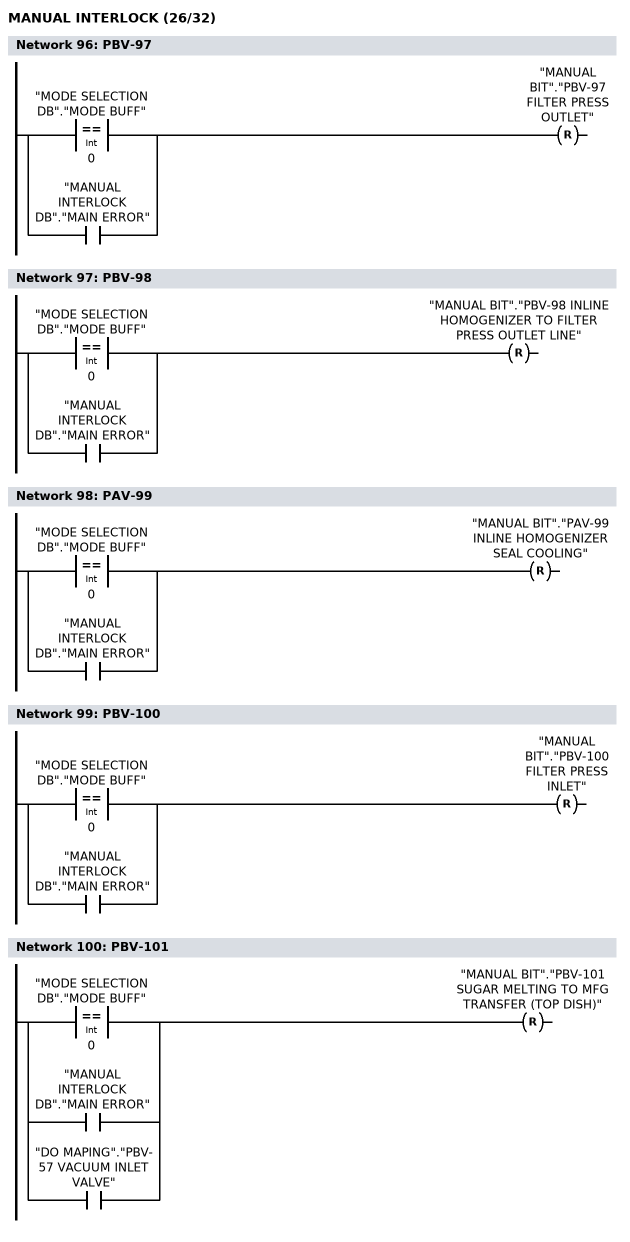
   RUNG wire#powerrail
      { S7_Templates := "SrcType := Int" } EQ_Contact(in1 := "MODE SELECTION DB"."MODE BUFF", in2 := 0)
      wire#w1
      R_Coil( "MANUAL BIT"."PBV-97 FILTER PRESS OUTLET" )
   END_RUNG
   RUNG wire#powerrail
      Contact( "MANUAL INTERLOCK DB"."MAIN ERROR" )
   END_RUNG wire#w1
   // the same network as SCL:
   IF ("MODE SELECTION DB"."MODE BUFF" = 0) OR "MANUAL INTERLOCK DB"."MAIN ERROR" THEN
       "MANUAL BIT"."PBV-97 FILTER PRESS OUTLET" := FALSE;
   END_IF;
END_REGION

REGION Network 97: PBV-98
   RUNG wire#powerrail
      { S7_Templates := "SrcType := Int" } EQ_Contact(in1 := "MODE SELECTION DB"."MODE BUFF", in2 := 0)
      wire#w1
      R_Coil( "MANUAL BIT"."PBV-98 INLINE HOMOGENIZER TO FILTER PRESS OUTLET LINE" )
   END_RUNG
   RUNG wire#powerrail
      Contact( "MANUAL INTERLOCK DB"."MAIN ERROR" )
   END_RUNG wire#w1
   // the same network as SCL:
   IF ("MODE SELECTION DB"."MODE BUFF" = 0) OR "MANUAL INTERLOCK DB"."MAIN ERROR" THEN
       "MANUAL BIT"."PBV-98 INLINE HOMOGENIZER TO FILTER PRESS OUTLET LINE" := FALSE;
   END_IF;
END_REGION

REGION Network 98: PAV-99
   RUNG wire#powerrail
      { S7_Templates := "SrcType := Int" } EQ_Contact(in1 := "MODE SELECTION DB"."MODE BUFF", in2 := 0)
      wire#w1
      R_Coil( "MANUAL BIT"."PAV-99 INLINE HOMOGENIZER SEAL COOLING" )
   END_RUNG
   RUNG wire#powerrail
      Contact( "MANUAL INTERLOCK DB"."MAIN ERROR" )
   END_RUNG wire#w1
   // the same network as SCL:
   IF ("MODE SELECTION DB"."MODE BUFF" = 0) OR "MANUAL INTERLOCK DB"."MAIN ERROR" THEN
       "MANUAL BIT"."PAV-99 INLINE HOMOGENIZER SEAL COOLING" := FALSE;
   END_IF;
END_REGION

REGION Network 99: PBV-100
   RUNG wire#powerrail
      { S7_Templates := "SrcType := Int" } EQ_Contact(in1 := "MODE SELECTION DB"."MODE BUFF", in2 := 0)
      wire#w1
      R_Coil( "MANUAL BIT"."PBV-100 FILTER PRESS INLET" )
   END_RUNG
   RUNG wire#powerrail
      Contact( "MANUAL INTERLOCK DB"."MAIN ERROR" )
   END_RUNG wire#w1
   // the same network as SCL:
   IF ("MODE SELECTION DB"."MODE BUFF" = 0) OR "MANUAL INTERLOCK DB"."MAIN ERROR" THEN
       "MANUAL BIT"."PBV-100 FILTER PRESS INLET" := FALSE;
   END_IF;
END_REGION

REGION Network 100: PBV-101
   RUNG wire#powerrail
      { S7_Templates := "SrcType := Int" } EQ_Contact(in1 := "MODE SELECTION DB"."MODE BUFF", in2 := 0)
      wire#w1
      R_Coil( "MANUAL BIT"."PBV-101 SUGAR MELTING TO MFG TRANSFER (TOP DISH)" )
   END_RUNG
   RUNG wire#powerrail
      Contact( "MANUAL INTERLOCK DB"."MAIN ERROR" )
   END_RUNG wire#w1
   RUNG wire#powerrail
      Contact( "DO MAPING"."PBV-57 VACUUM INLET VALVE" )
   END_RUNG wire#w1
   // the same network as SCL:
   IF ("MODE SELECTION DB"."MODE BUFF" = 0) OR "MANUAL INTERLOCK DB"."MAIN ERROR" OR "DO MAPING"."PBV-57 VACUUM INLET VALVE" THEN
       "MANUAL BIT"."PBV-101 SUGAR MELTING TO MFG TRANSFER (TOP DISH)" := FALSE;
   END_IF;
END_REGION

REGION Network 101: PBV-102
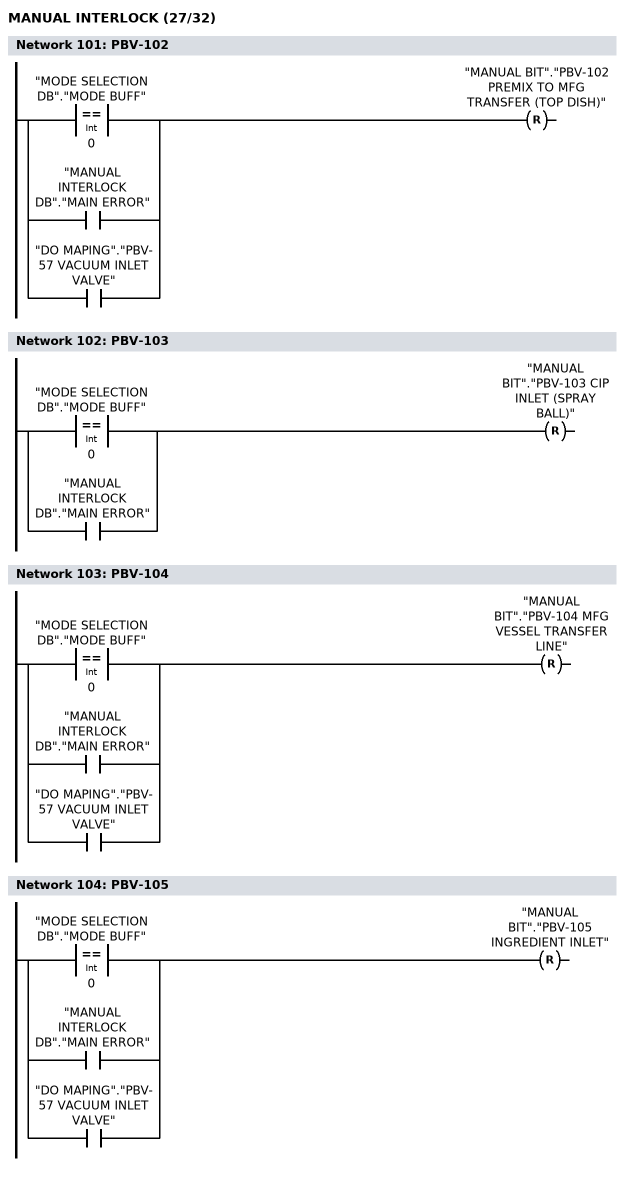
   RUNG wire#powerrail
      { S7_Templates := "SrcType := Int" } EQ_Contact(in1 := "MODE SELECTION DB"."MODE BUFF", in2 := 0)
      wire#w1
      R_Coil( "MANUAL BIT"."PBV-102 PREMIX TO MFG TRANSFER (TOP DISH)" )
   END_RUNG
   RUNG wire#powerrail
      Contact( "MANUAL INTERLOCK DB"."MAIN ERROR" )
   END_RUNG wire#w1
   RUNG wire#powerrail
      Contact( "DO MAPING"."PBV-57 VACUUM INLET VALVE" )
   END_RUNG wire#w1
   // the same network as SCL:
   IF ("MODE SELECTION DB"."MODE BUFF" = 0) OR "MANUAL INTERLOCK DB"."MAIN ERROR" OR "DO MAPING"."PBV-57 VACUUM INLET VALVE" THEN
       "MANUAL BIT"."PBV-102 PREMIX TO MFG TRANSFER (TOP DISH)" := FALSE;
   END_IF;
END_REGION

REGION Network 102: PBV-103
   RUNG wire#powerrail
      { S7_Templates := "SrcType := Int" } EQ_Contact(in1 := "MODE SELECTION DB"."MODE BUFF", in2 := 0)
      wire#w1
      R_Coil( "MANUAL BIT"."PBV-103 CIP INLET (SPRAY BALL)" )
   END_RUNG
   RUNG wire#powerrail
      Contact( "MANUAL INTERLOCK DB"."MAIN ERROR" )
   END_RUNG wire#w1
   // the same network as SCL:
   IF ("MODE SELECTION DB"."MODE BUFF" = 0) OR "MANUAL INTERLOCK DB"."MAIN ERROR" THEN
       "MANUAL BIT"."PBV-103 CIP INLET (SPRAY BALL)" := FALSE;
   END_IF;
END_REGION

REGION Network 103: PBV-104
   RUNG wire#powerrail
      { S7_Templates := "SrcType := Int" } EQ_Contact(in1 := "MODE SELECTION DB"."MODE BUFF", in2 := 0)
      wire#w1
      R_Coil( "MANUAL BIT"."PBV-104 MFG VESSEL TRANSFER LINE" )
   END_RUNG
   RUNG wire#powerrail
      Contact( "MANUAL INTERLOCK DB"."MAIN ERROR" )
   END_RUNG wire#w1
   RUNG wire#powerrail
      Contact( "DO MAPING"."PBV-57 VACUUM INLET VALVE" )
   END_RUNG wire#w1
   // the same network as SCL:
   IF ("MODE SELECTION DB"."MODE BUFF" = 0) OR "MANUAL INTERLOCK DB"."MAIN ERROR" OR "DO MAPING"."PBV-57 VACUUM INLET VALVE" THEN
       "MANUAL BIT"."PBV-104 MFG VESSEL TRANSFER LINE" := FALSE;
   END_IF;
END_REGION

REGION Network 104: PBV-105
   RUNG wire#powerrail
      { S7_Templates := "SrcType := Int" } EQ_Contact(in1 := "MODE SELECTION DB"."MODE BUFF", in2 := 0)
      wire#w1
      R_Coil( "MANUAL BIT"."PBV-105 INGREDIENT INLET" )
   END_RUNG
   RUNG wire#powerrail
      Contact( "MANUAL INTERLOCK DB"."MAIN ERROR" )
   END_RUNG wire#w1
   RUNG wire#powerrail
      Contact( "DO MAPING"."PBV-57 VACUUM INLET VALVE" )
   END_RUNG wire#w1
   // the same network as SCL:
   IF ("MODE SELECTION DB"."MODE BUFF" = 0) OR "MANUAL INTERLOCK DB"."MAIN ERROR" OR "DO MAPING"."PBV-57 VACUUM INLET VALVE" THEN
       "MANUAL BIT"."PBV-105 INGREDIENT INLET" := FALSE;
   END_IF;
END_REGION

REGION Network 105: PBV-106
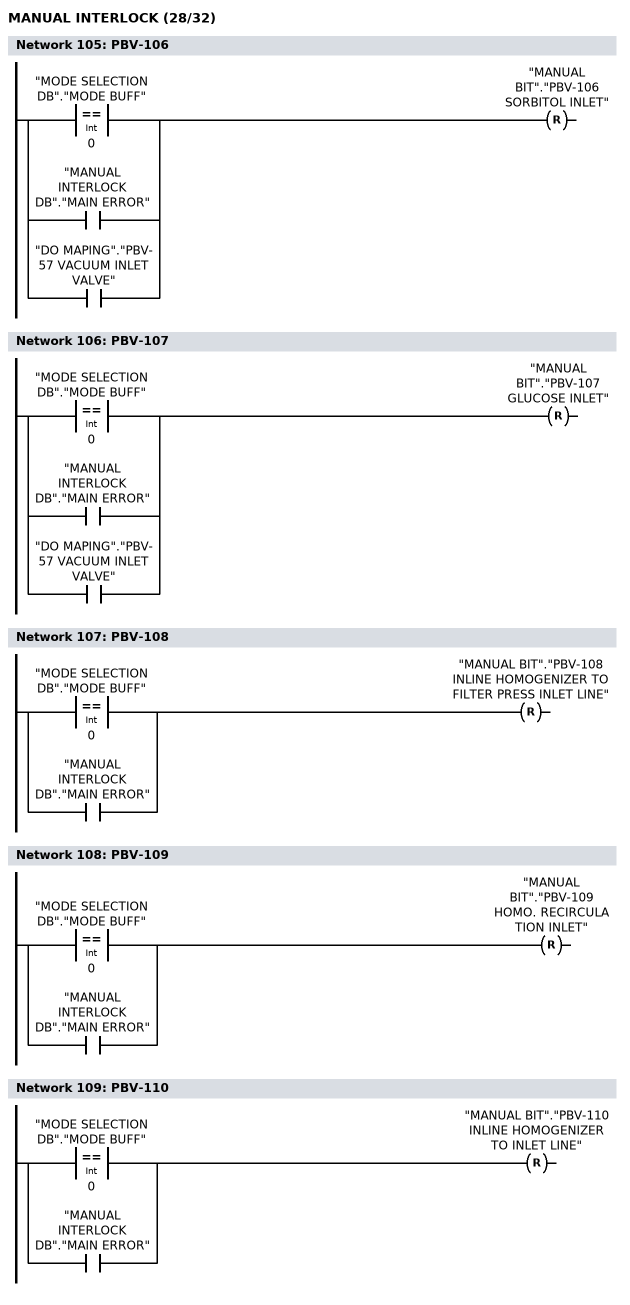
   RUNG wire#powerrail
      { S7_Templates := "SrcType := Int" } EQ_Contact(in1 := "MODE SELECTION DB"."MODE BUFF", in2 := 0)
      wire#w1
      R_Coil( "MANUAL BIT"."PBV-106 SORBITOL INLET" )
   END_RUNG
   RUNG wire#powerrail
      Contact( "MANUAL INTERLOCK DB"."MAIN ERROR" )
   END_RUNG wire#w1
   RUNG wire#powerrail
      Contact( "DO MAPING"."PBV-57 VACUUM INLET VALVE" )
   END_RUNG wire#w1
   // the same network as SCL:
   IF ("MODE SELECTION DB"."MODE BUFF" = 0) OR "MANUAL INTERLOCK DB"."MAIN ERROR" OR "DO MAPING"."PBV-57 VACUUM INLET VALVE" THEN
       "MANUAL BIT"."PBV-106 SORBITOL INLET" := FALSE;
   END_IF;
END_REGION

REGION Network 106: PBV-107
   RUNG wire#powerrail
      { S7_Templates := "SrcType := Int" } EQ_Contact(in1 := "MODE SELECTION DB"."MODE BUFF", in2 := 0)
      wire#w1
      R_Coil( "MANUAL BIT"."PBV-107 GLUCOSE INLET" )
   END_RUNG
   RUNG wire#powerrail
      Contact( "MANUAL INTERLOCK DB"."MAIN ERROR" )
   END_RUNG wire#w1
   RUNG wire#powerrail
      Contact( "DO MAPING"."PBV-57 VACUUM INLET VALVE" )
   END_RUNG wire#w1
   // the same network as SCL:
   IF ("MODE SELECTION DB"."MODE BUFF" = 0) OR "MANUAL INTERLOCK DB"."MAIN ERROR" OR "DO MAPING"."PBV-57 VACUUM INLET VALVE" THEN
       "MANUAL BIT"."PBV-107 GLUCOSE INLET" := FALSE;
   END_IF;
END_REGION

REGION Network 107: PBV-108
   RUNG wire#powerrail
      { S7_Templates := "SrcType := Int" } EQ_Contact(in1 := "MODE SELECTION DB"."MODE BUFF", in2 := 0)
      wire#w1
      R_Coil( "MANUAL BIT"."PBV-108 INLINE HOMOGENIZER TO FILTER PRESS INLET LINE" )
   END_RUNG
   RUNG wire#powerrail
      Contact( "MANUAL INTERLOCK DB"."MAIN ERROR" )
   END_RUNG wire#w1
   // the same network as SCL:
   IF ("MODE SELECTION DB"."MODE BUFF" = 0) OR "MANUAL INTERLOCK DB"."MAIN ERROR" THEN
       "MANUAL BIT"."PBV-108 INLINE HOMOGENIZER TO FILTER PRESS INLET LINE" := FALSE;
   END_IF;
END_REGION

REGION Network 108: PBV-109
   RUNG wire#powerrail
      { S7_Templates := "SrcType := Int" } EQ_Contact(in1 := "MODE SELECTION DB"."MODE BUFF", in2 := 0)
      wire#w1
      R_Coil( "MANUAL BIT"."PBV-109 HOMO. RECIRCULATION INLET" )
   END_RUNG
   RUNG wire#powerrail
      Contact( "MANUAL INTERLOCK DB"."MAIN ERROR" )
   END_RUNG wire#w1
   // the same network as SCL:
   IF ("MODE SELECTION DB"."MODE BUFF" = 0) OR "MANUAL INTERLOCK DB"."MAIN ERROR" THEN
       "MANUAL BIT"."PBV-109 HOMO. RECIRCULATION INLET" := FALSE;
   END_IF;
END_REGION

REGION Network 109: PBV-110
   RUNG wire#powerrail
      { S7_Templates := "SrcType := Int" } EQ_Contact(in1 := "MODE SELECTION DB"."MODE BUFF", in2 := 0)
      wire#w1
      R_Coil( "MANUAL BIT"."PBV-110 INLINE HOMOGENIZER TO INLET LINE" )
   END_RUNG
   RUNG wire#powerrail
      Contact( "MANUAL INTERLOCK DB"."MAIN ERROR" )
   END_RUNG wire#w1
   // the same network as SCL:
   IF ("MODE SELECTION DB"."MODE BUFF" = 0) OR "MANUAL INTERLOCK DB"."MAIN ERROR" THEN
       "MANUAL BIT"."PBV-110 INLINE HOMOGENIZER TO INLET LINE" := FALSE;
   END_IF;
END_REGION

REGION Network 110: PBV-111
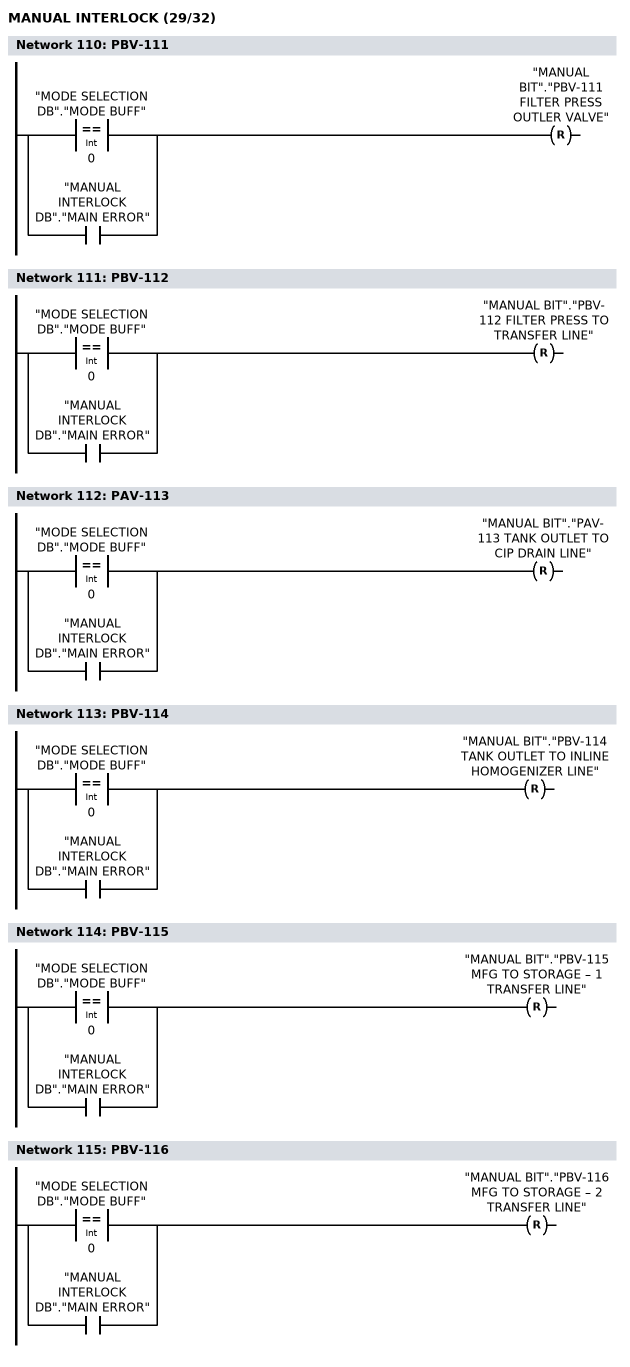
   RUNG wire#powerrail
      { S7_Templates := "SrcType := Int" } EQ_Contact(in1 := "MODE SELECTION DB"."MODE BUFF", in2 := 0)
      wire#w1
      R_Coil( "MANUAL BIT"."PBV-111 FILTER PRESS OUTLER VALVE" )
   END_RUNG
   RUNG wire#powerrail
      Contact( "MANUAL INTERLOCK DB"."MAIN ERROR" )
   END_RUNG wire#w1
   // the same network as SCL:
   IF ("MODE SELECTION DB"."MODE BUFF" = 0) OR "MANUAL INTERLOCK DB"."MAIN ERROR" THEN
       "MANUAL BIT"."PBV-111 FILTER PRESS OUTLER VALVE" := FALSE;
   END_IF;
END_REGION

REGION Network 111: PBV-112
   RUNG wire#powerrail
      { S7_Templates := "SrcType := Int" } EQ_Contact(in1 := "MODE SELECTION DB"."MODE BUFF", in2 := 0)
      wire#w1
      R_Coil( "MANUAL BIT"."PBV-112 FILTER PRESS TO TRANSFER LINE" )
   END_RUNG
   RUNG wire#powerrail
      Contact( "MANUAL INTERLOCK DB"."MAIN ERROR" )
   END_RUNG wire#w1
   // the same network as SCL:
   IF ("MODE SELECTION DB"."MODE BUFF" = 0) OR "MANUAL INTERLOCK DB"."MAIN ERROR" THEN
       "MANUAL BIT"."PBV-112 FILTER PRESS TO TRANSFER LINE" := FALSE;
   END_IF;
END_REGION

REGION Network 112: PAV-113
   RUNG wire#powerrail
      { S7_Templates := "SrcType := Int" } EQ_Contact(in1 := "MODE SELECTION DB"."MODE BUFF", in2 := 0)
      wire#w1
      R_Coil( "MANUAL BIT"."PAV-113 TANK OUTLET TO CIP DRAIN LINE" )
   END_RUNG
   RUNG wire#powerrail
      Contact( "MANUAL INTERLOCK DB"."MAIN ERROR" )
   END_RUNG wire#w1
   // the same network as SCL:
   IF ("MODE SELECTION DB"."MODE BUFF" = 0) OR "MANUAL INTERLOCK DB"."MAIN ERROR" THEN
       "MANUAL BIT"."PAV-113 TANK OUTLET TO CIP DRAIN LINE" := FALSE;
   END_IF;
END_REGION

REGION Network 113: PBV-114
   RUNG wire#powerrail
      { S7_Templates := "SrcType := Int" } EQ_Contact(in1 := "MODE SELECTION DB"."MODE BUFF", in2 := 0)
      wire#w1
      R_Coil( "MANUAL BIT"."PBV-114 TANK OUTLET TO INLINE HOMOGENIZER LINE" )
   END_RUNG
   RUNG wire#powerrail
      Contact( "MANUAL INTERLOCK DB"."MAIN ERROR" )
   END_RUNG wire#w1
   // the same network as SCL:
   IF ("MODE SELECTION DB"."MODE BUFF" = 0) OR "MANUAL INTERLOCK DB"."MAIN ERROR" THEN
       "MANUAL BIT"."PBV-114 TANK OUTLET TO INLINE HOMOGENIZER LINE" := FALSE;
   END_IF;
END_REGION

REGION Network 114: PBV-115
   RUNG wire#powerrail
      { S7_Templates := "SrcType := Int" } EQ_Contact(in1 := "MODE SELECTION DB"."MODE BUFF", in2 := 0)
      wire#w1
      R_Coil( "MANUAL BIT"."PBV-115 MFG TO STORAGE – 1 TRANSFER LINE" )
   END_RUNG
   RUNG wire#powerrail
      Contact( "MANUAL INTERLOCK DB"."MAIN ERROR" )
   END_RUNG wire#w1
   // the same network as SCL:
   IF ("MODE SELECTION DB"."MODE BUFF" = 0) OR "MANUAL INTERLOCK DB"."MAIN ERROR" THEN
       "MANUAL BIT"."PBV-115 MFG TO STORAGE – 1 TRANSFER LINE" := FALSE;
   END_IF;
END_REGION

REGION Network 115: PBV-116
   RUNG wire#powerrail
      { S7_Templates := "SrcType := Int" } EQ_Contact(in1 := "MODE SELECTION DB"."MODE BUFF", in2 := 0)
      wire#w1
      R_Coil( "MANUAL BIT"."PBV-116 MFG TO STORAGE – 2 TRANSFER LINE" )
   END_RUNG
   RUNG wire#powerrail
      Contact( "MANUAL INTERLOCK DB"."MAIN ERROR" )
   END_RUNG wire#w1
   // the same network as SCL:
   IF ("MODE SELECTION DB"."MODE BUFF" = 0) OR "MANUAL INTERLOCK DB"."MAIN ERROR" THEN
       "MANUAL BIT"."PBV-116 MFG TO STORAGE – 2 TRANSFER LINE" := FALSE;
   END_IF;
END_REGION

REGION Network 116: PBV-117
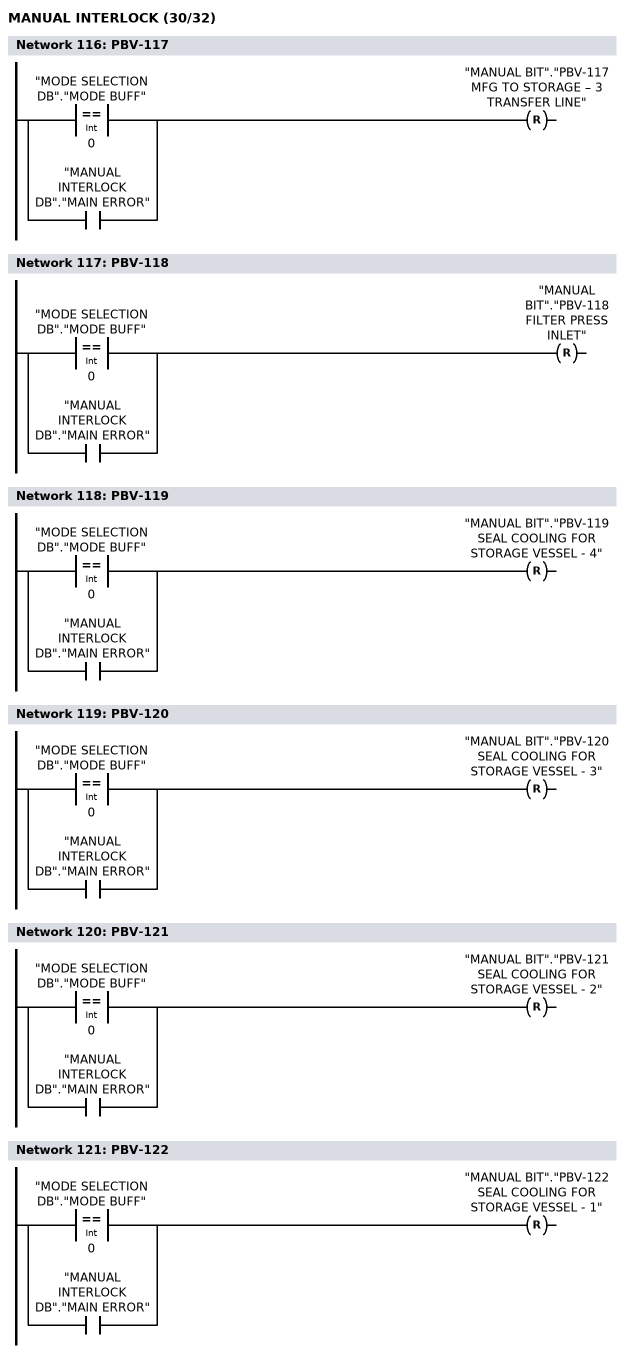
   RUNG wire#powerrail
      { S7_Templates := "SrcType := Int" } EQ_Contact(in1 := "MODE SELECTION DB"."MODE BUFF", in2 := 0)
      wire#w1
      R_Coil( "MANUAL BIT"."PBV-117 MFG TO STORAGE – 3 TRANSFER LINE" )
   END_RUNG
   RUNG wire#powerrail
      Contact( "MANUAL INTERLOCK DB"."MAIN ERROR" )
   END_RUNG wire#w1
   // the same network as SCL:
   IF ("MODE SELECTION DB"."MODE BUFF" = 0) OR "MANUAL INTERLOCK DB"."MAIN ERROR" THEN
       "MANUAL BIT"."PBV-117 MFG TO STORAGE – 3 TRANSFER LINE" := FALSE;
   END_IF;
END_REGION

REGION Network 117: PBV-118
   RUNG wire#powerrail
      { S7_Templates := "SrcType := Int" } EQ_Contact(in1 := "MODE SELECTION DB"."MODE BUFF", in2 := 0)
      wire#w1
      R_Coil( "MANUAL BIT"."PBV-118 FILTER PRESS INLET" )
   END_RUNG
   RUNG wire#powerrail
      Contact( "MANUAL INTERLOCK DB"."MAIN ERROR" )
   END_RUNG wire#w1
   // the same network as SCL:
   IF ("MODE SELECTION DB"."MODE BUFF" = 0) OR "MANUAL INTERLOCK DB"."MAIN ERROR" THEN
       "MANUAL BIT"."PBV-118 FILTER PRESS INLET" := FALSE;
   END_IF;
END_REGION

REGION Network 118: PBV-119
   RUNG wire#powerrail
      { S7_Templates := "SrcType := Int" } EQ_Contact(in1 := "MODE SELECTION DB"."MODE BUFF", in2 := 0)
      wire#w1
      R_Coil( "MANUAL BIT"."PBV-119 SEAL COOLING FOR STORAGE VESSEL - 4" )
   END_RUNG
   RUNG wire#powerrail
      Contact( "MANUAL INTERLOCK DB"."MAIN ERROR" )
   END_RUNG wire#w1
   // the same network as SCL:
   IF ("MODE SELECTION DB"."MODE BUFF" = 0) OR "MANUAL INTERLOCK DB"."MAIN ERROR" THEN
       "MANUAL BIT"."PBV-119 SEAL COOLING FOR STORAGE VESSEL - 4" := FALSE;
   END_IF;
END_REGION

REGION Network 119: PBV-120
   RUNG wire#powerrail
      { S7_Templates := "SrcType := Int" } EQ_Contact(in1 := "MODE SELECTION DB"."MODE BUFF", in2 := 0)
      wire#w1
      R_Coil( "MANUAL BIT"."PBV-120 SEAL COOLING FOR STORAGE VESSEL - 3" )
   END_RUNG
   RUNG wire#powerrail
      Contact( "MANUAL INTERLOCK DB"."MAIN ERROR" )
   END_RUNG wire#w1
   // the same network as SCL:
   IF ("MODE SELECTION DB"."MODE BUFF" = 0) OR "MANUAL INTERLOCK DB"."MAIN ERROR" THEN
       "MANUAL BIT"."PBV-120 SEAL COOLING FOR STORAGE VESSEL - 3" := FALSE;
   END_IF;
END_REGION

REGION Network 120: PBV-121
   RUNG wire#powerrail
      { S7_Templates := "SrcType := Int" } EQ_Contact(in1 := "MODE SELECTION DB"."MODE BUFF", in2 := 0)
      wire#w1
      R_Coil( "MANUAL BIT"."PBV-121 SEAL COOLING FOR STORAGE VESSEL - 2" )
   END_RUNG
   RUNG wire#powerrail
      Contact( "MANUAL INTERLOCK DB"."MAIN ERROR" )
   END_RUNG wire#w1
   // the same network as SCL:
   IF ("MODE SELECTION DB"."MODE BUFF" = 0) OR "MANUAL INTERLOCK DB"."MAIN ERROR" THEN
       "MANUAL BIT"."PBV-121 SEAL COOLING FOR STORAGE VESSEL - 2" := FALSE;
   END_IF;
END_REGION

REGION Network 121: PBV-122
   RUNG wire#powerrail
      { S7_Templates := "SrcType := Int" } EQ_Contact(in1 := "MODE SELECTION DB"."MODE BUFF", in2 := 0)
      wire#w1
      R_Coil( "MANUAL BIT"."PBV-122 SEAL COOLING FOR STORAGE VESSEL - 1" )
   END_RUNG
   RUNG wire#powerrail
      Contact( "MANUAL INTERLOCK DB"."MAIN ERROR" )
   END_RUNG wire#w1
   // the same network as SCL:
   IF ("MODE SELECTION DB"."MODE BUFF" = 0) OR "MANUAL INTERLOCK DB"."MAIN ERROR" THEN
       "MANUAL BIT"."PBV-122 SEAL COOLING FOR STORAGE VESSEL - 1" := FALSE;
   END_IF;
END_REGION

REGION Network 122: PBV-123
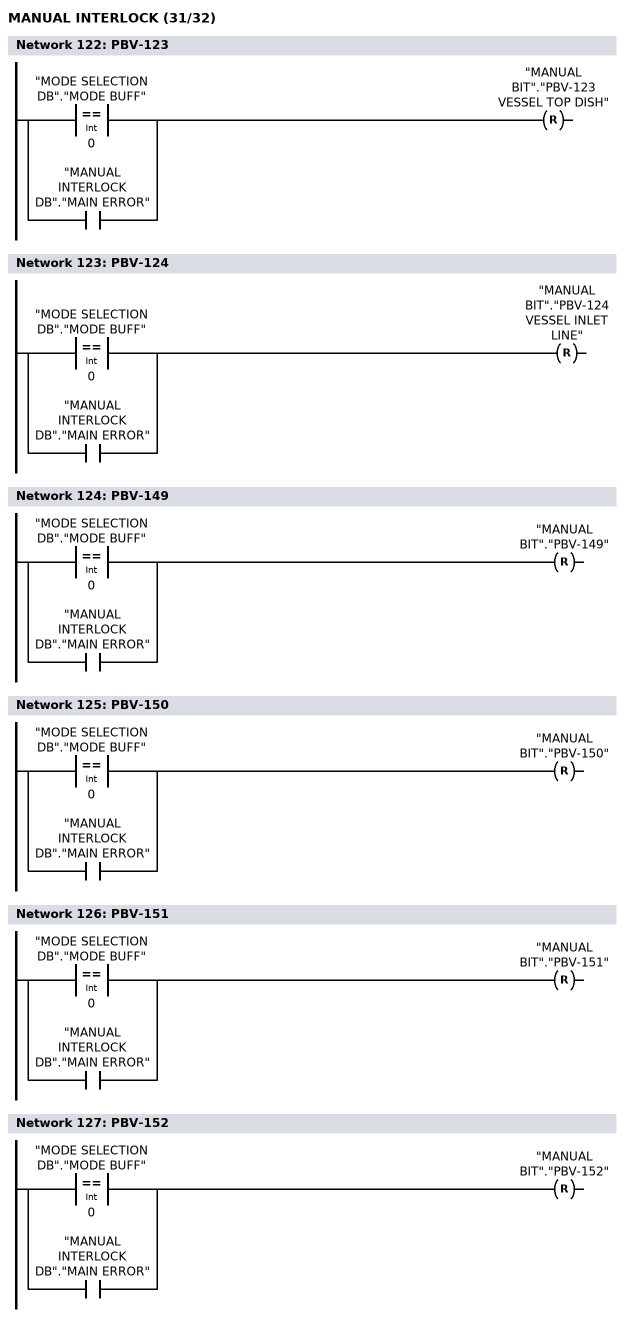
   RUNG wire#powerrail
      { S7_Templates := "SrcType := Int" } EQ_Contact(in1 := "MODE SELECTION DB"."MODE BUFF", in2 := 0)
      wire#w1
      R_Coil( "MANUAL BIT"."PBV-123 VESSEL TOP DISH" )
   END_RUNG
   RUNG wire#powerrail
      Contact( "MANUAL INTERLOCK DB"."MAIN ERROR" )
   END_RUNG wire#w1
   // the same network as SCL:
   IF ("MODE SELECTION DB"."MODE BUFF" = 0) OR "MANUAL INTERLOCK DB"."MAIN ERROR" THEN
       "MANUAL BIT"."PBV-123 VESSEL TOP DISH" := FALSE;
   END_IF;
END_REGION

REGION Network 123: PBV-124
   RUNG wire#powerrail
      { S7_Templates := "SrcType := Int" } EQ_Contact(in1 := "MODE SELECTION DB"."MODE BUFF", in2 := 0)
      wire#w1
      R_Coil( "MANUAL BIT"."PBV-124 VESSEL INLET LINE" )
   END_RUNG
   RUNG wire#powerrail
      Contact( "MANUAL INTERLOCK DB"."MAIN ERROR" )
   END_RUNG wire#w1
   // the same network as SCL:
   IF ("MODE SELECTION DB"."MODE BUFF" = 0) OR "MANUAL INTERLOCK DB"."MAIN ERROR" THEN
       "MANUAL BIT"."PBV-124 VESSEL INLET LINE" := FALSE;
   END_IF;
END_REGION

REGION Network 124: PBV-149
   RUNG wire#powerrail
      { S7_Templates := "SrcType := Int" } EQ_Contact(in1 := "MODE SELECTION DB"."MODE BUFF", in2 := 0)
      wire#w1
      R_Coil( "MANUAL BIT"."PBV-149" )
   END_RUNG
   RUNG wire#powerrail
      Contact( "MANUAL INTERLOCK DB"."MAIN ERROR" )
   END_RUNG wire#w1
   // the same network as SCL:
   IF ("MODE SELECTION DB"."MODE BUFF" = 0) OR "MANUAL INTERLOCK DB"."MAIN ERROR" THEN
       "MANUAL BIT"."PBV-149" := FALSE;
   END_IF;
END_REGION

REGION Network 125: PBV-150
   RUNG wire#powerrail
      { S7_Templates := "SrcType := Int" } EQ_Contact(in1 := "MODE SELECTION DB"."MODE BUFF", in2 := 0)
      wire#w1
      R_Coil( "MANUAL BIT"."PBV-150" )
   END_RUNG
   RUNG wire#powerrail
      Contact( "MANUAL INTERLOCK DB"."MAIN ERROR" )
   END_RUNG wire#w1
   // the same network as SCL:
   IF ("MODE SELECTION DB"."MODE BUFF" = 0) OR "MANUAL INTERLOCK DB"."MAIN ERROR" THEN
       "MANUAL BIT"."PBV-150" := FALSE;
   END_IF;
END_REGION

REGION Network 126: PBV-151
   RUNG wire#powerrail
      { S7_Templates := "SrcType := Int" } EQ_Contact(in1 := "MODE SELECTION DB"."MODE BUFF", in2 := 0)
      wire#w1
      R_Coil( "MANUAL BIT"."PBV-151" )
   END_RUNG
   RUNG wire#powerrail
      Contact( "MANUAL INTERLOCK DB"."MAIN ERROR" )
   END_RUNG wire#w1
   // the same network as SCL:
   IF ("MODE SELECTION DB"."MODE BUFF" = 0) OR "MANUAL INTERLOCK DB"."MAIN ERROR" THEN
       "MANUAL BIT"."PBV-151" := FALSE;
   END_IF;
END_REGION

REGION Network 127: PBV-152
   RUNG wire#powerrail
      { S7_Templates := "SrcType := Int" } EQ_Contact(in1 := "MODE SELECTION DB"."MODE BUFF", in2 := 0)
      wire#w1
      R_Coil( "MANUAL BIT"."PBV-152" )
   END_RUNG
   RUNG wire#powerrail
      Contact( "MANUAL INTERLOCK DB"."MAIN ERROR" )
   END_RUNG wire#w1
   // the same network as SCL:
   IF ("MODE SELECTION DB"."MODE BUFF" = 0) OR "MANUAL INTERLOCK DB"."MAIN ERROR" THEN
       "MANUAL BIT"."PBV-152" := FALSE;
   END_IF;
END_REGION

REGION Network 128: PBV-153
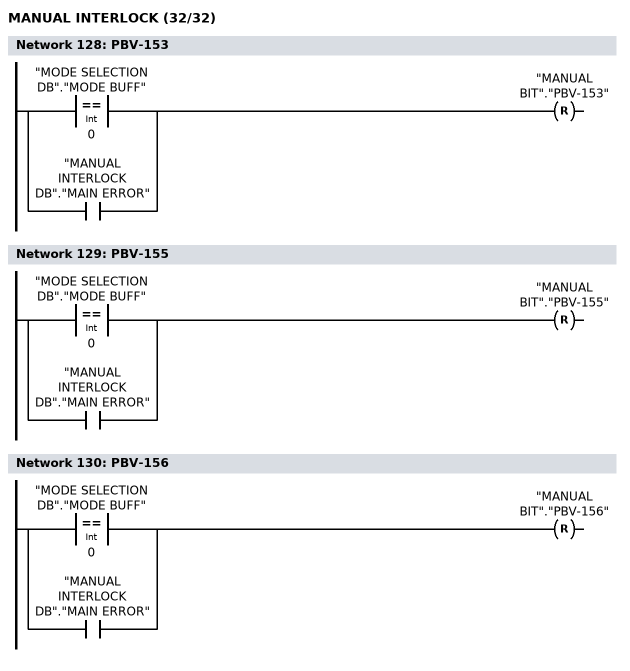
   RUNG wire#powerrail
      { S7_Templates := "SrcType := Int" } EQ_Contact(in1 := "MODE SELECTION DB"."MODE BUFF", in2 := 0)
      wire#w1
      R_Coil( "MANUAL BIT"."PBV-153" )
   END_RUNG
   RUNG wire#powerrail
      Contact( "MANUAL INTERLOCK DB"."MAIN ERROR" )
   END_RUNG wire#w1
   // the same network as SCL:
   IF ("MODE SELECTION DB"."MODE BUFF" = 0) OR "MANUAL INTERLOCK DB"."MAIN ERROR" THEN
       "MANUAL BIT"."PBV-153" := FALSE;
   END_IF;
END_REGION

REGION Network 129: PBV-155
   RUNG wire#powerrail
      { S7_Templates := "SrcType := Int" } EQ_Contact(in1 := "MODE SELECTION DB"."MODE BUFF", in2 := 0)
      wire#w1
      R_Coil( "MANUAL BIT"."PBV-155" )
   END_RUNG
   RUNG wire#powerrail
      Contact( "MANUAL INTERLOCK DB"."MAIN ERROR" )
   END_RUNG wire#w1
   // the same network as SCL:
   IF ("MODE SELECTION DB"."MODE BUFF" = 0) OR "MANUAL INTERLOCK DB"."MAIN ERROR" THEN
       "MANUAL BIT"."PBV-155" := FALSE;
   END_IF;
END_REGION

REGION Network 130: PBV-156
   RUNG wire#powerrail
      { S7_Templates := "SrcType := Int" } EQ_Contact(in1 := "MODE SELECTION DB"."MODE BUFF", in2 := 0)
      wire#w1
      R_Coil( "MANUAL BIT"."PBV-156" )
   END_RUNG
   RUNG wire#powerrail
      Contact( "MANUAL INTERLOCK DB"."MAIN ERROR" )
   END_RUNG wire#w1
   // the same network as SCL:
   IF ("MODE SELECTION DB"."MODE BUFF" = 0) OR "MANUAL INTERLOCK DB"."MAIN ERROR" THEN
       "MANUAL BIT"."PBV-156" := FALSE;
   END_IF;
END_REGION
END_FUNCTION

FUNCTION "TEMP CUTOFF LOGIC" : Void   // FC11, LAD
{ S7_Optimized_Access := 'TRUE' }
// stored: SetENOAutomatically false
   VAR_TEMP   // added for the SCL form of the ladder/FBD networks
      _w1 : Bool;
      _w2 : Bool;
   END_VAR
BEGIN

REGION Network 1: MFG_TEMP. VALUE ///////////////////////////////////////////////////////////////
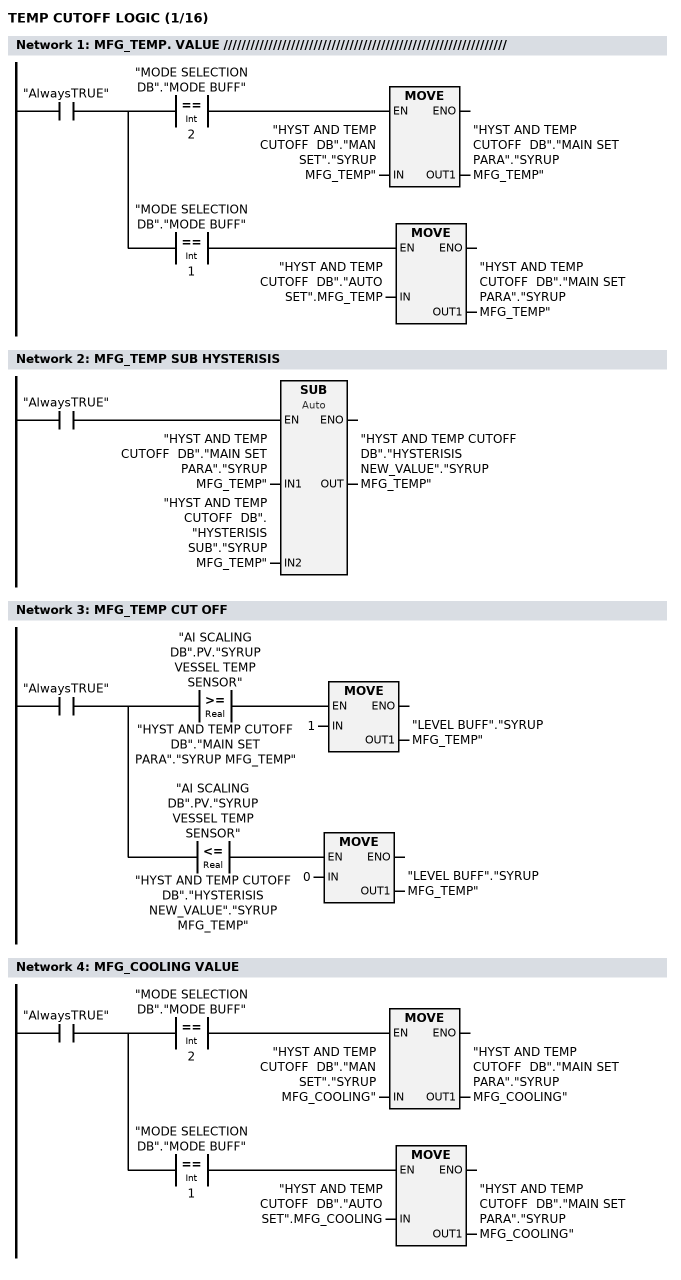
   RUNG wire#powerrail
      Contact( "AlwaysTRUE" )
      wire#w1
      { S7_Templates := "SrcType := Int" } EQ_Contact(in1 := "MODE SELECTION DB"."MODE BUFF", in2 := 2)
      Move(in := "HYST AND TEMP CUTOFF  DB"."MAN SET"."SYRUP MFG_TEMP", out1 => "HYST AND TEMP CUTOFF  DB"."MAIN SET PARA"."SYRUP MFG_TEMP")
   END_RUNG
   RUNG wire#w1
      { S7_Templates := "SrcType := Int" } EQ_Contact(in1 := "MODE SELECTION DB"."MODE BUFF", in2 := 1)
      Move(in := "HYST AND TEMP CUTOFF  DB"."AUTO SET".MFG_TEMP, out1 => "HYST AND TEMP CUTOFF  DB"."MAIN SET PARA"."SYRUP MFG_TEMP")
   END_RUNG
   // the same network as SCL:
   IF "AlwaysTRUE" AND ("MODE SELECTION DB"."MODE BUFF" = 2) THEN
       "HYST AND TEMP CUTOFF  DB"."MAIN SET PARA"."SYRUP MFG_TEMP" := "HYST AND TEMP CUTOFF  DB"."MAN SET"."SYRUP MFG_TEMP";
   END_IF;
   IF "AlwaysTRUE" AND ("MODE SELECTION DB"."MODE BUFF" = 1) THEN
       "HYST AND TEMP CUTOFF  DB"."MAIN SET PARA"."SYRUP MFG_TEMP" := "HYST AND TEMP CUTOFF  DB"."AUTO SET".MFG_TEMP;
   END_IF;
END_REGION

REGION Network 2: MFG_TEMP SUB HYSTERISIS
   RUNG wire#powerrail
      Contact( "AlwaysTRUE" )
      Sub(in1 := "HYST AND TEMP CUTOFF  DB"."MAIN SET PARA"."SYRUP MFG_TEMP", in2 := "HYST AND TEMP CUTOFF  DB"."HYSTERISIS SUB"."SYRUP MFG_TEMP", out => "HYST AND TEMP CUTOFF  DB"."HYSTERISIS NEW_VALUE"."SYRUP MFG_TEMP")
   END_RUNG
   // the same network as SCL:
   IF "AlwaysTRUE" THEN
       "HYST AND TEMP CUTOFF  DB"."HYSTERISIS NEW_VALUE"."SYRUP MFG_TEMP" := "HYST AND TEMP CUTOFF  DB"."MAIN SET PARA"."SYRUP MFG_TEMP" - "HYST AND TEMP CUTOFF  DB"."HYSTERISIS SUB"."SYRUP MFG_TEMP";
   END_IF;
END_REGION

REGION Network 3: MFG_TEMP CUT OFF
   RUNG wire#powerrail
      Contact( "AlwaysTRUE" )
      wire#w1
      { S7_Templates := "SrcType := Real" } GE_Contact(in1 := "AI SCALING DB".PV."SYRUP VESSEL TEMP SENSOR", in2 := "HYST AND TEMP CUTOFF  DB"."MAIN SET PARA"."SYRUP MFG_TEMP")
      Move(in := 1, out1 => "LEVEL BUFF"."SYRUP MFG_TEMP")
   END_RUNG
   RUNG wire#w1
      { S7_Templates := "SrcType := Real" } LE_Contact(in1 := "AI SCALING DB".PV."SYRUP VESSEL TEMP SENSOR", in2 := "HYST AND TEMP CUTOFF  DB"."HYSTERISIS NEW_VALUE"."SYRUP MFG_TEMP")
      Move(in := 0, out1 => "LEVEL BUFF"."SYRUP MFG_TEMP")
   END_RUNG
   // the same network as SCL:
   IF "AlwaysTRUE" AND ("AI SCALING DB".PV."SYRUP VESSEL TEMP SENSOR" >= "HYST AND TEMP CUTOFF  DB"."MAIN SET PARA"."SYRUP MFG_TEMP") THEN
       "LEVEL BUFF"."SYRUP MFG_TEMP" := 1;
   END_IF;
   IF "AlwaysTRUE" AND ("AI SCALING DB".PV."SYRUP VESSEL TEMP SENSOR" <= "HYST AND TEMP CUTOFF  DB"."HYSTERISIS NEW_VALUE"."SYRUP MFG_TEMP") THEN
       "LEVEL BUFF"."SYRUP MFG_TEMP" := 0;
   END_IF;
END_REGION

REGION Network 4: MFG_COOLING VALUE
   RUNG wire#powerrail
      Contact( "AlwaysTRUE" )
      wire#w1
      { S7_Templates := "SrcType := Int" } EQ_Contact(in1 := "MODE SELECTION DB"."MODE BUFF", in2 := 2)
      Move(in := "HYST AND TEMP CUTOFF  DB"."MAN SET"."SYRUP MFG_COOLING", out1 => "HYST AND TEMP CUTOFF  DB"."MAIN SET PARA"."SYRUP MFG_COOLING")
   END_RUNG
   RUNG wire#w1
      { S7_Templates := "SrcType := Int" } EQ_Contact(in1 := "MODE SELECTION DB"."MODE BUFF", in2 := 1)
      Move(in := "HYST AND TEMP CUTOFF  DB"."AUTO SET".MFG_COOLING, out1 => "HYST AND TEMP CUTOFF  DB"."MAIN SET PARA"."SYRUP MFG_COOLING")
   END_RUNG
   // the same network as SCL:
   IF "AlwaysTRUE" AND ("MODE SELECTION DB"."MODE BUFF" = 2) THEN
       "HYST AND TEMP CUTOFF  DB"."MAIN SET PARA"."SYRUP MFG_COOLING" := "HYST AND TEMP CUTOFF  DB"."MAN SET"."SYRUP MFG_COOLING";
   END_IF;
   IF "AlwaysTRUE" AND ("MODE SELECTION DB"."MODE BUFF" = 1) THEN
       "HYST AND TEMP CUTOFF  DB"."MAIN SET PARA"."SYRUP MFG_COOLING" := "HYST AND TEMP CUTOFF  DB"."AUTO SET".MFG_COOLING;
   END_IF;
END_REGION

REGION Network 5: MFG_COOLING SUB HYSTERISIS
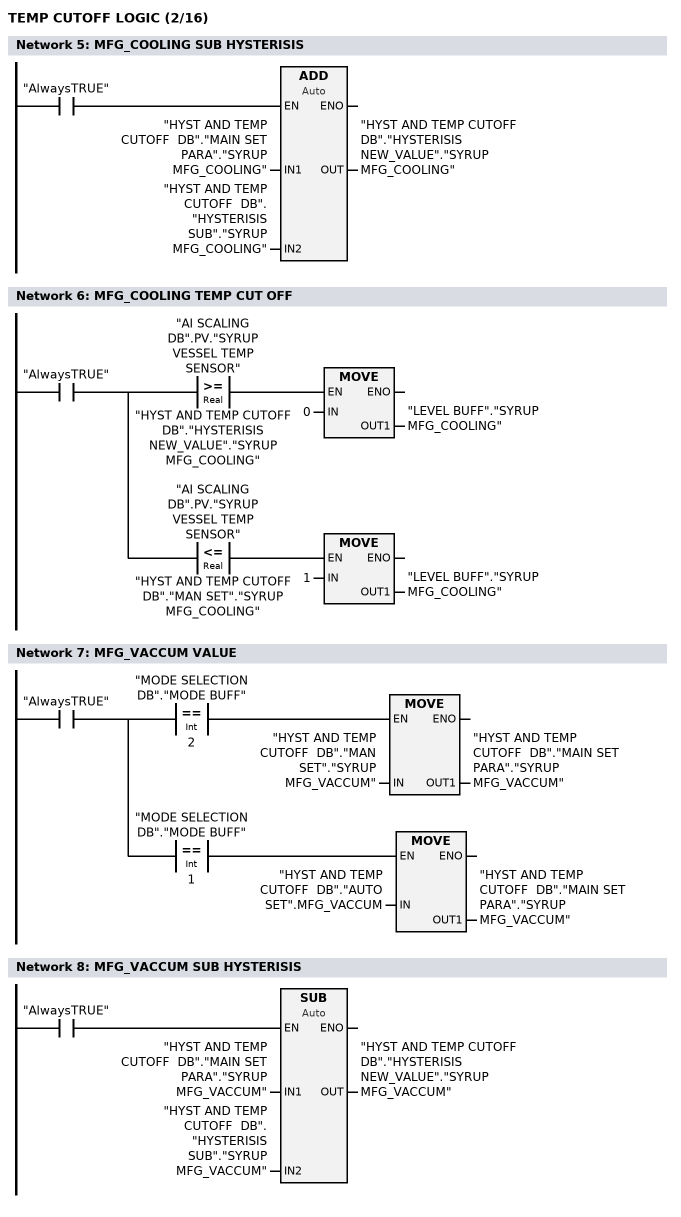
   RUNG wire#powerrail
      Contact( "AlwaysTRUE" )
      Add(in1 := "HYST AND TEMP CUTOFF  DB"."MAIN SET PARA"."SYRUP MFG_COOLING", in2 := "HYST AND TEMP CUTOFF  DB"."HYSTERISIS SUB"."SYRUP MFG_COOLING", out => "HYST AND TEMP CUTOFF  DB"."HYSTERISIS NEW_VALUE"."SYRUP MFG_COOLING")
   END_RUNG
   // the same network as SCL:
   IF "AlwaysTRUE" THEN
       "HYST AND TEMP CUTOFF  DB"."HYSTERISIS NEW_VALUE"."SYRUP MFG_COOLING" := "HYST AND TEMP CUTOFF  DB"."MAIN SET PARA"."SYRUP MFG_COOLING" + "HYST AND TEMP CUTOFF  DB"."HYSTERISIS SUB"."SYRUP MFG_COOLING";
   END_IF;
END_REGION

REGION Network 6: MFG_COOLING TEMP CUT OFF
   RUNG wire#powerrail
      Contact( "AlwaysTRUE" )
      wire#w1
      { S7_Templates := "SrcType := Real" } GE_Contact(in1 := "AI SCALING DB".PV."SYRUP VESSEL TEMP SENSOR", in2 := "HYST AND TEMP CUTOFF  DB"."HYSTERISIS NEW_VALUE"."SYRUP MFG_COOLING")
      Move(in := 0, out1 => "LEVEL BUFF"."SYRUP MFG_COOLING")
   END_RUNG
   RUNG wire#w1
      { S7_Templates := "SrcType := Real" } LE_Contact(in1 := "AI SCALING DB".PV."SYRUP VESSEL TEMP SENSOR", in2 := "HYST AND TEMP CUTOFF  DB"."MAN SET"."SYRUP MFG_COOLING")
      Move(in := 1, out1 => "LEVEL BUFF"."SYRUP MFG_COOLING")
   END_RUNG
   // the same network as SCL:
   IF "AlwaysTRUE" AND ("AI SCALING DB".PV."SYRUP VESSEL TEMP SENSOR" >= "HYST AND TEMP CUTOFF  DB"."HYSTERISIS NEW_VALUE"."SYRUP MFG_COOLING") THEN
       "LEVEL BUFF"."SYRUP MFG_COOLING" := 0;
   END_IF;
   IF "AlwaysTRUE" AND ("AI SCALING DB".PV."SYRUP VESSEL TEMP SENSOR" <= "HYST AND TEMP CUTOFF  DB"."MAN SET"."SYRUP MFG_COOLING") THEN
       "LEVEL BUFF"."SYRUP MFG_COOLING" := 1;
   END_IF;
END_REGION

REGION Network 7: MFG_VACCUM VALUE
   RUNG wire#powerrail
      Contact( "AlwaysTRUE" )
      wire#w1
      { S7_Templates := "SrcType := Int" } EQ_Contact(in1 := "MODE SELECTION DB"."MODE BUFF", in2 := 2)
      Move(in := "HYST AND TEMP CUTOFF  DB"."MAN SET"."SYRUP MFG_VACCUM", out1 => "HYST AND TEMP CUTOFF  DB"."MAIN SET PARA"."SYRUP MFG_VACCUM")
   END_RUNG
   RUNG wire#w1
      { S7_Templates := "SrcType := Int" } EQ_Contact(in1 := "MODE SELECTION DB"."MODE BUFF", in2 := 1)
      Move(in := "HYST AND TEMP CUTOFF  DB"."AUTO SET".MFG_VACCUM, out1 => "HYST AND TEMP CUTOFF  DB"."MAIN SET PARA"."SYRUP MFG_VACCUM")
   END_RUNG
   // the same network as SCL:
   IF "AlwaysTRUE" AND ("MODE SELECTION DB"."MODE BUFF" = 2) THEN
       "HYST AND TEMP CUTOFF  DB"."MAIN SET PARA"."SYRUP MFG_VACCUM" := "HYST AND TEMP CUTOFF  DB"."MAN SET"."SYRUP MFG_VACCUM";
   END_IF;
   IF "AlwaysTRUE" AND ("MODE SELECTION DB"."MODE BUFF" = 1) THEN
       "HYST AND TEMP CUTOFF  DB"."MAIN SET PARA"."SYRUP MFG_VACCUM" := "HYST AND TEMP CUTOFF  DB"."AUTO SET".MFG_VACCUM;
   END_IF;
END_REGION

REGION Network 8: MFG_VACCUM SUB HYSTERISIS
   RUNG wire#powerrail
      Contact( "AlwaysTRUE" )
      Sub(in1 := "HYST AND TEMP CUTOFF  DB"."MAIN SET PARA"."SYRUP MFG_VACCUM", in2 := "HYST AND TEMP CUTOFF  DB"."HYSTERISIS SUB"."SYRUP MFG_VACCUM", out => "HYST AND TEMP CUTOFF  DB"."HYSTERISIS NEW_VALUE"."SYRUP MFG_VACCUM")
   END_RUNG
   // the same network as SCL:
   IF "AlwaysTRUE" THEN
       "HYST AND TEMP CUTOFF  DB"."HYSTERISIS NEW_VALUE"."SYRUP MFG_VACCUM" := "HYST AND TEMP CUTOFF  DB"."MAIN SET PARA"."SYRUP MFG_VACCUM" - "HYST AND TEMP CUTOFF  DB"."HYSTERISIS SUB"."SYRUP MFG_VACCUM";
   END_IF;
END_REGION

REGION Network 9: MFG_VACCUM CUT OFF
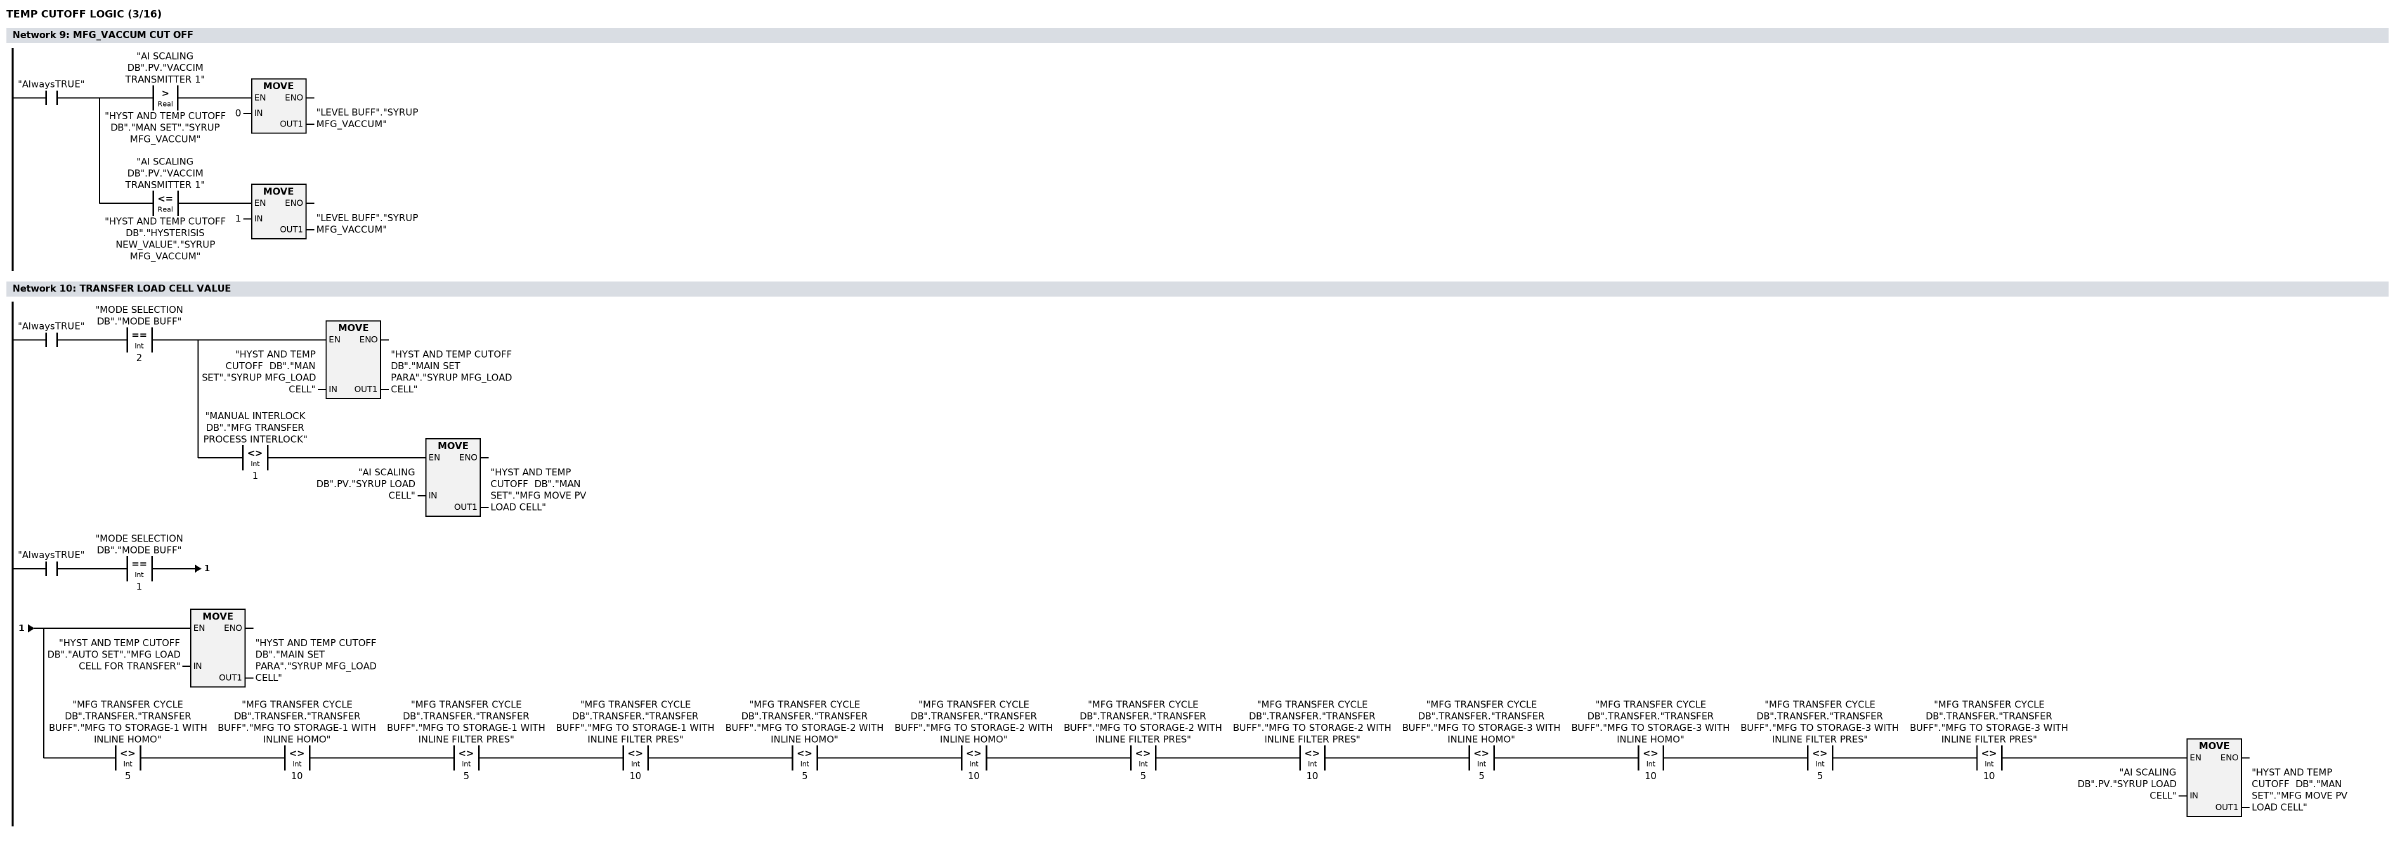
   RUNG wire#powerrail
      Contact( "AlwaysTRUE" )
      wire#w1
      { S7_Templates := "SrcType := Real" } GT_Contact(in1 := "AI SCALING DB".PV."VACCIM TRANSMITTER 1", in2 := "HYST AND TEMP CUTOFF  DB"."MAN SET"."SYRUP MFG_VACCUM")
      Move(in := 0, out1 => "LEVEL BUFF"."SYRUP MFG_VACCUM")
   END_RUNG
   RUNG wire#w1
      { S7_Templates := "SrcType := Real" } LE_Contact(in1 := "AI SCALING DB".PV."VACCIM TRANSMITTER 1", in2 := "HYST AND TEMP CUTOFF  DB"."HYSTERISIS NEW_VALUE"."SYRUP MFG_VACCUM")
      Move(in := 1, out1 => "LEVEL BUFF"."SYRUP MFG_VACCUM")
   END_RUNG
   // the same network as SCL:
   IF "AlwaysTRUE" AND ("AI SCALING DB".PV."VACCIM TRANSMITTER 1" > "HYST AND TEMP CUTOFF  DB"."MAN SET"."SYRUP MFG_VACCUM") THEN
       "LEVEL BUFF"."SYRUP MFG_VACCUM" := 0;
   END_IF;
   IF "AlwaysTRUE" AND ("AI SCALING DB".PV."VACCIM TRANSMITTER 1" <= "HYST AND TEMP CUTOFF  DB"."HYSTERISIS NEW_VALUE"."SYRUP MFG_VACCUM") THEN
       "LEVEL BUFF"."SYRUP MFG_VACCUM" := 1;
   END_IF;
END_REGION

REGION Network 10: TRANSFER LOAD CELL VALUE
   RUNG wire#powerrail
      Contact( "AlwaysTRUE" )
      { S7_Templates := "SrcType := Int" } EQ_Contact(in1 := "MODE SELECTION DB"."MODE BUFF", in2 := 2)
      wire#w1
      Move(in := "HYST AND TEMP CUTOFF  DB"."MAN SET"."SYRUP MFG_LOAD CELL", out1 => "HYST AND TEMP CUTOFF  DB"."MAIN SET PARA"."SYRUP MFG_LOAD CELL")
   END_RUNG
   RUNG wire#w1
      { S7_Templates := "SrcType := Int" } NE_Contact(in1 := "MANUAL INTERLOCK DB"."MFG TRANSFER PROCESS INTERLOCK", in2 := 1)
      Move(in := "AI SCALING DB".PV."SYRUP LOAD CELL", out1 => "HYST AND TEMP CUTOFF  DB"."MAN SET"."MFG MOVE PV LOAD CELL")
   END_RUNG
   RUNG wire#powerrail
      Contact( "AlwaysTRUE" )
      { S7_Templates := "SrcType := Int" } EQ_Contact(in1 := "MODE SELECTION DB"."MODE BUFF", in2 := 1)
      wire#w2
      Move(in := "HYST AND TEMP CUTOFF  DB"."AUTO SET"."MFG LOAD CELL FOR TRANSFER", out1 => "HYST AND TEMP CUTOFF  DB"."MAIN SET PARA"."SYRUP MFG_LOAD CELL")
   END_RUNG
   RUNG wire#w2
      { S7_Templates := "SrcType := Int" } NE_Contact(in1 := "MFG TRANSFER CYCLE DB".TRANSFER."TRANSFER BUFF"."MFG TO STORAGE-1 WITH INLINE HOMO", in2 := 5)
      { S7_Templates := "SrcType := Int" } NE_Contact(in1 := "MFG TRANSFER CYCLE DB".TRANSFER."TRANSFER BUFF"."MFG TO STORAGE-1 WITH INLINE HOMO", in2 := 10)
      { S7_Templates := "SrcType := Int" } NE_Contact(in1 := "MFG TRANSFER CYCLE DB".TRANSFER."TRANSFER BUFF"."MFG TO STORAGE-1 WITH INLINE FILTER PRES", in2 := 5)
      { S7_Templates := "SrcType := Int" } NE_Contact(in1 := "MFG TRANSFER CYCLE DB".TRANSFER."TRANSFER BUFF"."MFG TO STORAGE-1 WITH INLINE FILTER PRES", in2 := 10)
      { S7_Templates := "SrcType := Int" } NE_Contact(in1 := "MFG TRANSFER CYCLE DB".TRANSFER."TRANSFER BUFF"."MFG TO STORAGE-2 WITH INLINE HOMO", in2 := 5)
      { S7_Templates := "SrcType := Int" } NE_Contact(in1 := "MFG TRANSFER CYCLE DB".TRANSFER."TRANSFER BUFF"."MFG TO STORAGE-2 WITH INLINE HOMO", in2 := 10)
      { S7_Templates := "SrcType := Int" } NE_Contact(in1 := "MFG TRANSFER CYCLE DB".TRANSFER."TRANSFER BUFF"."MFG TO STORAGE-2 WITH INLINE FILTER PRES", in2 := 5)
      { S7_Templates := "SrcType := Int" } NE_Contact(in1 := "MFG TRANSFER CYCLE DB".TRANSFER."TRANSFER BUFF"."MFG TO STORAGE-2 WITH INLINE FILTER PRES", in2 := 10)
      { S7_Templates := "SrcType := Int" } NE_Contact(in1 := "MFG TRANSFER CYCLE DB".TRANSFER."TRANSFER BUFF"."MFG TO STORAGE-3 WITH INLINE HOMO", in2 := 5)
      { S7_Templates := "SrcType := Int" } NE_Contact(in1 := "MFG TRANSFER CYCLE DB".TRANSFER."TRANSFER BUFF"."MFG TO STORAGE-3 WITH INLINE HOMO", in2 := 10)
      { S7_Templates := "SrcType := Int" } NE_Contact(in1 := "MFG TRANSFER CYCLE DB".TRANSFER."TRANSFER BUFF"."MFG TO STORAGE-3 WITH INLINE FILTER PRES", in2 := 5)
      { S7_Templates := "SrcType := Int" } NE_Contact(in1 := "MFG TRANSFER CYCLE DB".TRANSFER."TRANSFER BUFF"."MFG TO STORAGE-3 WITH INLINE FILTER PRES", in2 := 10)
      Move(in := "AI SCALING DB".PV."SYRUP LOAD CELL", out1 => "HYST AND TEMP CUTOFF  DB"."MAN SET"."MFG MOVE PV LOAD CELL")
   END_RUNG
   // the same network as SCL:
   #_w1 := "AlwaysTRUE" AND ("MODE SELECTION DB"."MODE BUFF" = 2);
   IF #_w1 THEN
       "HYST AND TEMP CUTOFF  DB"."MAIN SET PARA"."SYRUP MFG_LOAD CELL" := "HYST AND TEMP CUTOFF  DB"."MAN SET"."SYRUP MFG_LOAD CELL";
   END_IF;
   IF #_w1 AND ("MANUAL INTERLOCK DB"."MFG TRANSFER PROCESS INTERLOCK" <> 1) THEN
       "HYST AND TEMP CUTOFF  DB"."MAN SET"."MFG MOVE PV LOAD CELL" := "AI SCALING DB".PV."SYRUP LOAD CELL";
   END_IF;
   #_w2 := "AlwaysTRUE" AND ("MODE SELECTION DB"."MODE BUFF" = 1);
   IF #_w2 THEN
       "HYST AND TEMP CUTOFF  DB"."MAIN SET PARA"."SYRUP MFG_LOAD CELL" := "HYST AND TEMP CUTOFF  DB"."AUTO SET"."MFG LOAD CELL FOR TRANSFER";
   END_IF;
   IF #_w2 AND ("MFG TRANSFER CYCLE DB".TRANSFER."TRANSFER BUFF"."MFG TO STORAGE-1 WITH INLINE HOMO" <> 5) AND ("MFG TRANSFER CYCLE DB".TRANSFER."TRANSFER BUFF"."MFG TO STORAGE-1 WITH INLINE HOMO" <> 10) AND ("MFG TRANSFER CYCLE DB".TRANSFER."TRANSFER BUFF"."MFG TO STORAGE-1 WITH INLINE FILTER PRES" <> 5) AND ("MFG TRANSFER CYCLE DB".TRANSFER."TRANSFER BUFF"."MFG TO STORAGE-1 WITH INLINE FILTER PRES" <> 10) AND ("MFG TRANSFER CYCLE DB".TRANSFER."TRANSFER BUFF"."MFG TO STORAGE-2 WITH INLINE HOMO" <> 5) AND ("MFG TRANSFER CYCLE DB".TRANSFER."TRANSFER BUFF"."MFG TO STORAGE-2 WITH INLINE HOMO" <> 10) AND ("MFG TRANSFER CYCLE DB".TRANSFER."TRANSFER BUFF"."MFG TO STORAGE-2 WITH INLINE FILTER PRES" <> 5) AND ("MFG TRANSFER CYCLE DB".TRANSFER."TRANSFER BUFF"."MFG TO STORAGE-2 WITH INLINE FILTER PRES" <> 10) AND ("MFG TRANSFER CYCLE DB".TRANSFER."TRANSFER BUFF"."MFG TO STORAGE-3 WITH INLINE HOMO" <> 5) AND ("MFG TRANSFER CYCLE DB".TRANSFER."TRANSFER BUFF"."MFG TO STORAGE-3 WITH INLINE HOMO" <> 10) AND ("MFG TRANSFER CYCLE DB".TRANSFER."TRANSFER BUFF"."MFG TO STORAGE-3 WITH INLINE FILTER PRES" <> 5) AND ("MFG TRANSFER CYCLE DB".TRANSFER."TRANSFER BUFF"."MFG TO STORAGE-3 WITH INLINE FILTER PRES" <> 10) THEN
       "HYST AND TEMP CUTOFF  DB"."MAN SET"."MFG MOVE PV LOAD CELL" := "AI SCALING DB".PV."SYRUP LOAD CELL";
   END_IF;
END_REGION

REGION Network 11: TRANSFER CALCULATE
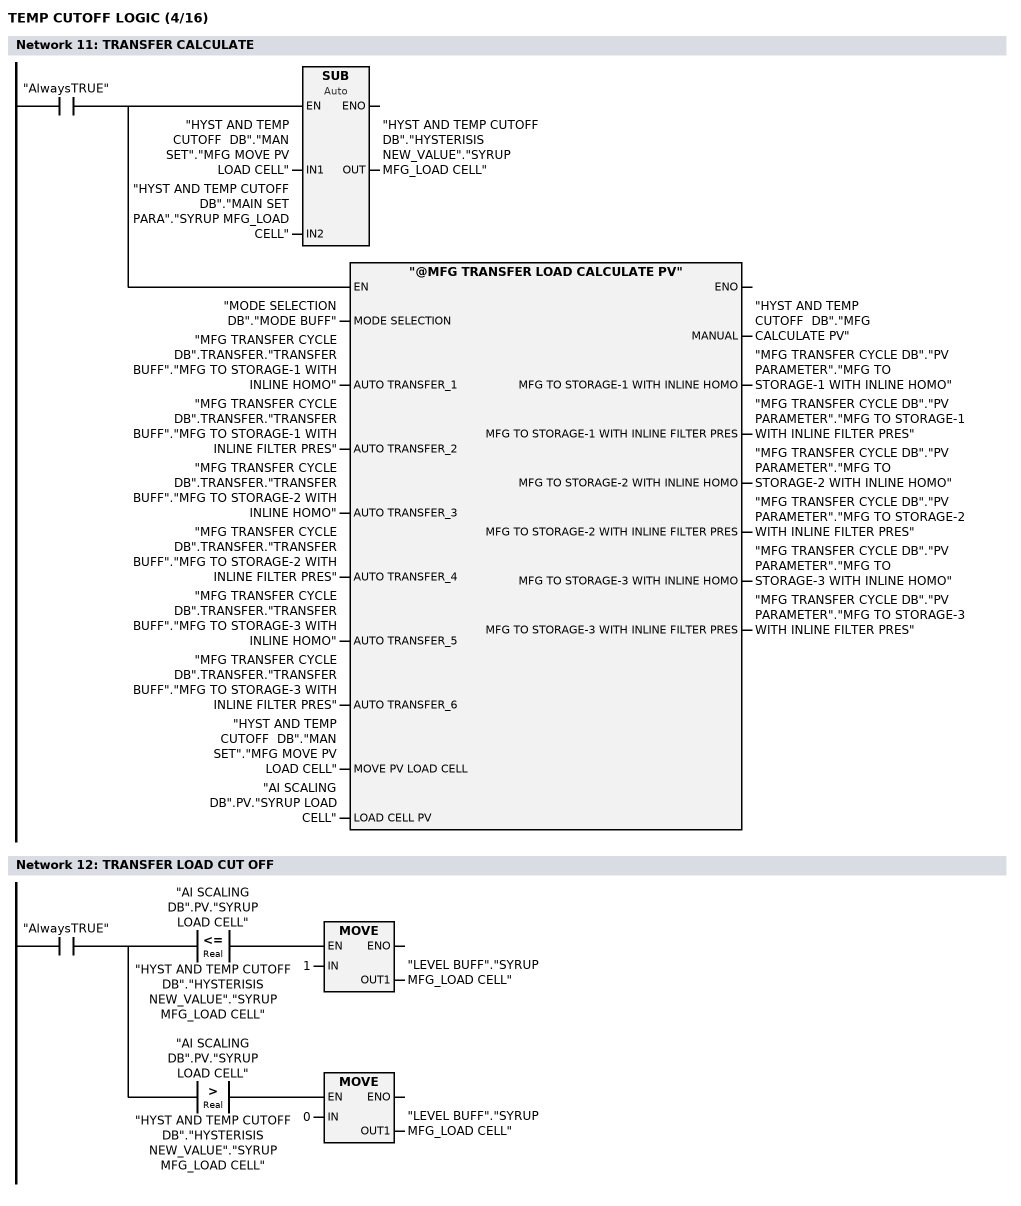
   RUNG wire#powerrail
      Contact( "AlwaysTRUE" )
      wire#w1
      Sub(in1 := "HYST AND TEMP CUTOFF  DB"."MAN SET"."MFG MOVE PV LOAD CELL", in2 := "HYST AND TEMP CUTOFF  DB"."MAIN SET PARA"."SYRUP MFG_LOAD CELL", out => "HYST AND TEMP CUTOFF  DB"."HYSTERISIS NEW_VALUE"."SYRUP MFG_LOAD CELL")
   END_RUNG
   RUNG wire#w1
      "@MFG TRANSFER LOAD CALCULATE PV"("MODE SELECTION" := "MODE SELECTION DB"."MODE BUFF", "AUTO TRANSFER_1" := "MFG TRANSFER CYCLE DB".TRANSFER."TRANSFER BUFF"."MFG TO STORAGE-1 WITH INLINE HOMO", "AUTO TRANSFER_2" := "MFG TRANSFER CYCLE DB".TRANSFER."TRANSFER BUFF"."MFG TO STORAGE-1 WITH INLINE FILTER PRES", "AUTO TRANSFER_3" := "MFG TRANSFER CYCLE DB".TRANSFER."TRANSFER BUFF"."MFG TO STORAGE-2 WITH INLINE HOMO", "AUTO TRANSFER_4" := "MFG TRANSFER CYCLE DB".TRANSFER."TRANSFER BUFF"."MFG TO STORAGE-2 WITH INLINE FILTER PRES", "AUTO TRANSFER_5" := "MFG TRANSFER CYCLE DB".TRANSFER."TRANSFER BUFF"."MFG TO STORAGE-3 WITH INLINE HOMO", "AUTO TRANSFER_6" := "MFG TRANSFER CYCLE DB".TRANSFER."TRANSFER BUFF"."MFG TO STORAGE-3 WITH INLINE FILTER PRES", "MOVE PV LOAD CELL" := "HYST AND TEMP CUTOFF  DB"."MAN SET"."MFG MOVE PV LOAD CELL", "LOAD CELL PV" := "AI SCALING DB".PV."SYRUP LOAD CELL", MANUAL => "HYST AND TEMP CUTOFF  DB"."MFG CALCULATE PV", "MFG TO STORAGE-1 WITH INLINE HOMO" => "MFG TRANSFER CYCLE DB"."PV PARAMETER"."MFG TO STORAGE-1 WITH INLINE HOMO", "MFG TO STORAGE-1 WITH INLINE FILTER PRES" => "MFG TRANSFER CYCLE DB"."PV PARAMETER"."MFG TO STORAGE-1 WITH INLINE FILTER PRES", "MFG TO STORAGE-2 WITH INLINE HOMO" => "MFG TRANSFER CYCLE DB"."PV PARAMETER"."MFG TO STORAGE-2 WITH INLINE HOMO", "MFG TO STORAGE-2 WITH INLINE FILTER PRES" => "MFG TRANSFER CYCLE DB"."PV PARAMETER"."MFG TO STORAGE-2 WITH INLINE FILTER PRES", "MFG TO STORAGE-3 WITH INLINE HOMO" => "MFG TRANSFER CYCLE DB"."PV PARAMETER"."MFG TO STORAGE-3 WITH INLINE HOMO", "MFG TO STORAGE-3 WITH INLINE FILTER PRES" => "MFG TRANSFER CYCLE DB"."PV PARAMETER"."MFG TO STORAGE-3 WITH INLINE FILTER PRES")
   END_RUNG
   // the same network as SCL:
   IF "AlwaysTRUE" THEN
       "HYST AND TEMP CUTOFF  DB"."HYSTERISIS NEW_VALUE"."SYRUP MFG_LOAD CELL" := "HYST AND TEMP CUTOFF  DB"."MAN SET"."MFG MOVE PV LOAD CELL" - "HYST AND TEMP CUTOFF  DB"."MAIN SET PARA"."SYRUP MFG_LOAD CELL";
       "@MFG TRANSFER LOAD CALCULATE PV"("MODE SELECTION" := "MODE SELECTION DB"."MODE BUFF",
                               "AUTO TRANSFER_1" := "MFG TRANSFER CYCLE DB".TRANSFER."TRANSFER BUFF"."MFG TO STORAGE-1 WITH INLINE HOMO",
                               "AUTO TRANSFER_2" := "MFG TRANSFER CYCLE DB".TRANSFER."TRANSFER BUFF"."MFG TO STORAGE-1 WITH INLINE FILTER PRES",
                               "AUTO TRANSFER_3" := "MFG TRANSFER CYCLE DB".TRANSFER."TRANSFER BUFF"."MFG TO STORAGE-2 WITH INLINE HOMO",
                               "AUTO TRANSFER_4" := "MFG TRANSFER CYCLE DB".TRANSFER."TRANSFER BUFF"."MFG TO STORAGE-2 WITH INLINE FILTER PRES",
                               "AUTO TRANSFER_5" := "MFG TRANSFER CYCLE DB".TRANSFER."TRANSFER BUFF"."MFG TO STORAGE-3 WITH INLINE HOMO",
                               "AUTO TRANSFER_6" := "MFG TRANSFER CYCLE DB".TRANSFER."TRANSFER BUFF"."MFG TO STORAGE-3 WITH INLINE FILTER PRES",
                               "MOVE PV LOAD CELL" := "HYST AND TEMP CUTOFF  DB"."MAN SET"."MFG MOVE PV LOAD CELL",
                               "LOAD CELL PV" := "AI SCALING DB".PV."SYRUP LOAD CELL",
                               MANUAL => "HYST AND TEMP CUTOFF  DB"."MFG CALCULATE PV",
                               "MFG TO STORAGE-1 WITH INLINE HOMO" => "MFG TRANSFER CYCLE DB"."PV PARAMETER"."MFG TO STORAGE-1 WITH INLINE HOMO",
                               "MFG TO STORAGE-1 WITH INLINE FILTER PRES" => "MFG TRANSFER CYCLE DB"."PV PARAMETER"."MFG TO STORAGE-1 WITH INLINE FILTER PRES",
                               "MFG TO STORAGE-2 WITH INLINE HOMO" => "MFG TRANSFER CYCLE DB"."PV PARAMETER"."MFG TO STORAGE-2 WITH INLINE HOMO",
                               "MFG TO STORAGE-2 WITH INLINE FILTER PRES" => "MFG TRANSFER CYCLE DB"."PV PARAMETER"."MFG TO STORAGE-2 WITH INLINE FILTER PRES",
                               "MFG TO STORAGE-3 WITH INLINE HOMO" => "MFG TRANSFER CYCLE DB"."PV PARAMETER"."MFG TO STORAGE-3 WITH INLINE HOMO",
                               "MFG TO STORAGE-3 WITH INLINE FILTER PRES" => "MFG TRANSFER CYCLE DB"."PV PARAMETER"."MFG TO STORAGE-3 WITH INLINE FILTER PRES");
   END_IF;
END_REGION

REGION Network 12: TRANSFER LOAD CUT OFF
   RUNG wire#powerrail
      Contact( "AlwaysTRUE" )
      wire#w1
      { S7_Templates := "SrcType := Real" } LE_Contact(in1 := "AI SCALING DB".PV."SYRUP LOAD CELL", in2 := "HYST AND TEMP CUTOFF  DB"."HYSTERISIS NEW_VALUE"."SYRUP MFG_LOAD CELL")
      Move(in := 1, out1 => "LEVEL BUFF"."SYRUP MFG_LOAD CELL")
   END_RUNG
   RUNG wire#w1
      { S7_Templates := "SrcType := Real" } GT_Contact(in1 := "AI SCALING DB".PV."SYRUP LOAD CELL", in2 := "HYST AND TEMP CUTOFF  DB"."HYSTERISIS NEW_VALUE"."SYRUP MFG_LOAD CELL")
      Move(in := 0, out1 => "LEVEL BUFF"."SYRUP MFG_LOAD CELL")
   END_RUNG
   // the same network as SCL:
   IF "AlwaysTRUE" AND ("AI SCALING DB".PV."SYRUP LOAD CELL" <= "HYST AND TEMP CUTOFF  DB"."HYSTERISIS NEW_VALUE"."SYRUP MFG_LOAD CELL") THEN
       "LEVEL BUFF"."SYRUP MFG_LOAD CELL" := 1;
   END_IF;
   IF "AlwaysTRUE" AND ("AI SCALING DB".PV."SYRUP LOAD CELL" > "HYST AND TEMP CUTOFF  DB"."HYSTERISIS NEW_VALUE"."SYRUP MFG_LOAD CELL") THEN
       "LEVEL BUFF"."SYRUP MFG_LOAD CELL" := 0;
   END_IF;
END_REGION

REGION Network 14: AUTO LOAD CELL VALUE
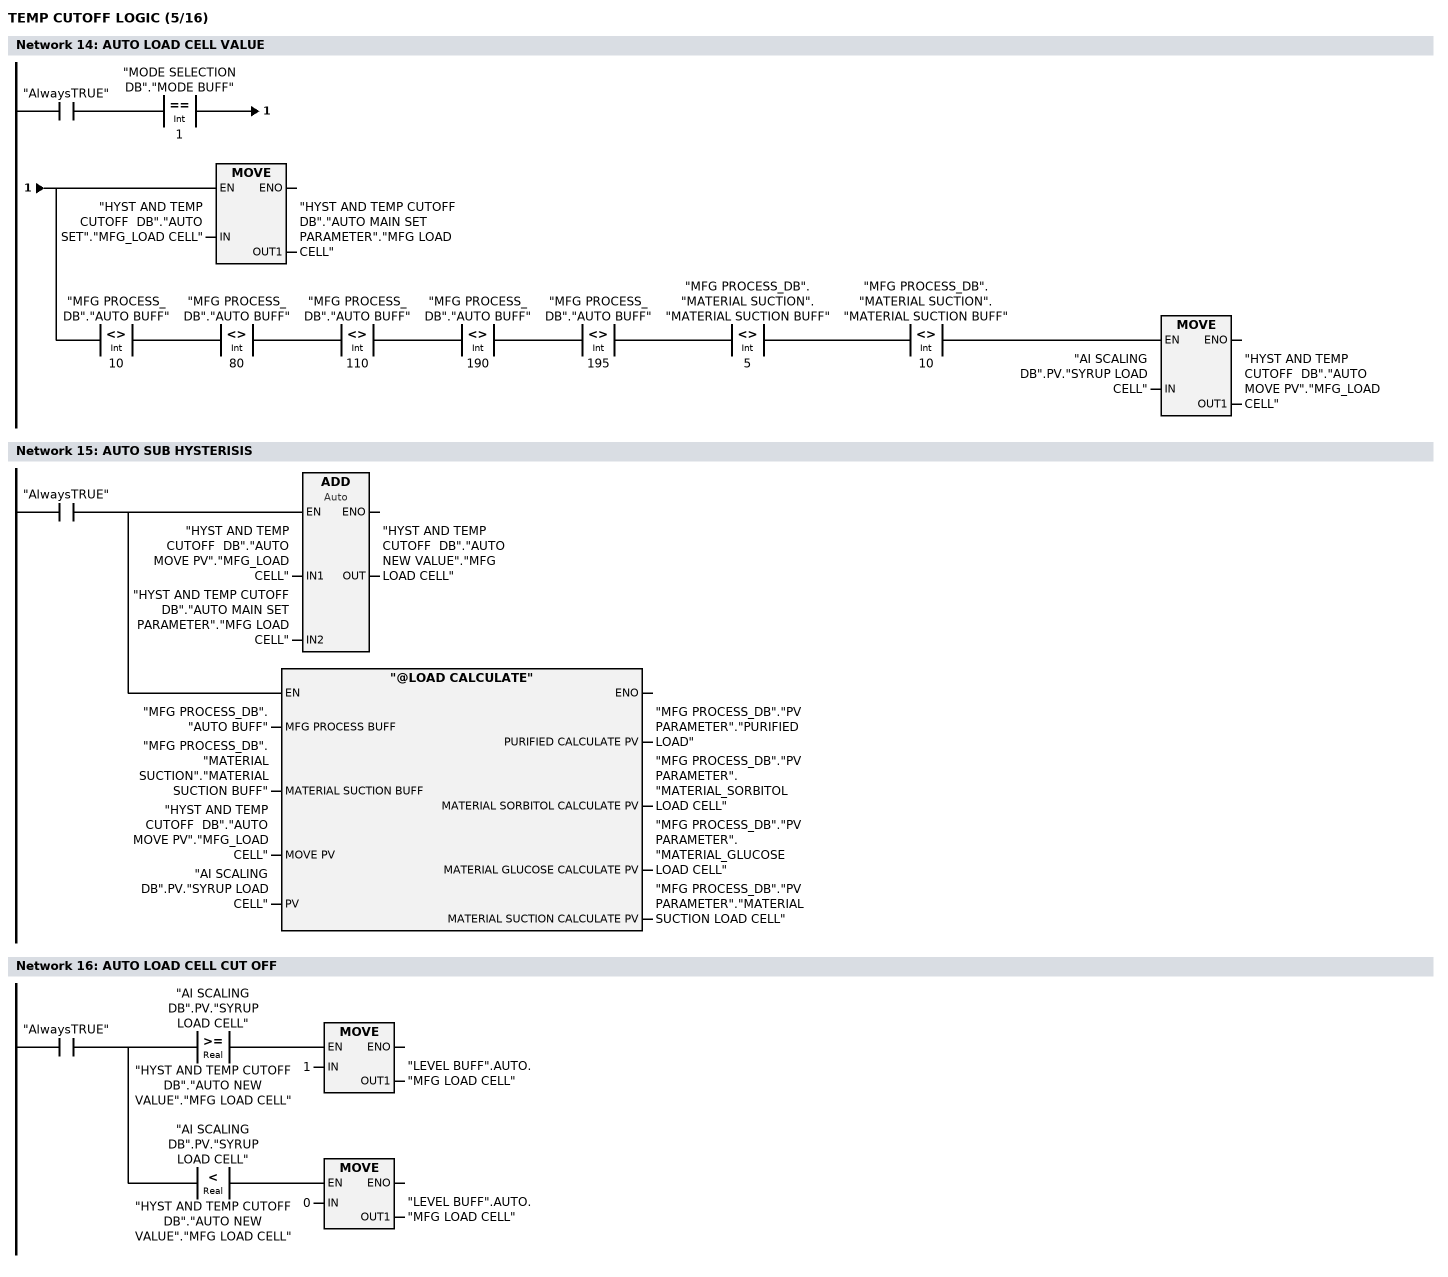
   RUNG wire#powerrail
      Contact( "AlwaysTRUE" )
      { S7_Templates := "SrcType := Int" } EQ_Contact(in1 := "MODE SELECTION DB"."MODE BUFF", in2 := 1)
      wire#w1
      Move(in := "HYST AND TEMP CUTOFF  DB"."AUTO SET"."MFG_LOAD CELL", out1 => "HYST AND TEMP CUTOFF  DB"."AUTO MAIN SET PARAMETER"."MFG LOAD CELL")
   END_RUNG
   RUNG wire#w1
      { S7_Templates := "SrcType := Int" } NE_Contact(in1 := "MFG PROCESS_DB"."AUTO BUFF", in2 := 10)
      { S7_Templates := "SrcType := Int" } NE_Contact(in1 := "MFG PROCESS_DB"."AUTO BUFF", in2 := 80)
      { S7_Templates := "SrcType := Int" } NE_Contact(in1 := "MFG PROCESS_DB"."AUTO BUFF", in2 := 110)
      { S7_Templates := "SrcType := Int" } NE_Contact(in1 := "MFG PROCESS_DB"."AUTO BUFF", in2 := 190)
      { S7_Templates := "SrcType := Int" } NE_Contact(in1 := "MFG PROCESS_DB"."AUTO BUFF", in2 := 195)
      { S7_Templates := "SrcType := Int" } NE_Contact(in1 := "MFG PROCESS_DB"."MATERIAL SUCTION"."MATERIAL SUCTION BUFF", in2 := 5)
      { S7_Templates := "SrcType := Int" } NE_Contact(in1 := "MFG PROCESS_DB"."MATERIAL SUCTION"."MATERIAL SUCTION BUFF", in2 := 10)
      Move(in := "AI SCALING DB".PV."SYRUP LOAD CELL", out1 => "HYST AND TEMP CUTOFF  DB"."AUTO MOVE PV"."MFG_LOAD CELL")
   END_RUNG
   // the same network as SCL:
   #_w1 := "AlwaysTRUE" AND ("MODE SELECTION DB"."MODE BUFF" = 1);
   IF #_w1 THEN
       "HYST AND TEMP CUTOFF  DB"."AUTO MAIN SET PARAMETER"."MFG LOAD CELL" := "HYST AND TEMP CUTOFF  DB"."AUTO SET"."MFG_LOAD CELL";
   END_IF;
   IF #_w1 AND ("MFG PROCESS_DB"."AUTO BUFF" <> 10) AND ("MFG PROCESS_DB"."AUTO BUFF" <> 80) AND ("MFG PROCESS_DB"."AUTO BUFF" <> 110) AND ("MFG PROCESS_DB"."AUTO BUFF" <> 190) AND ("MFG PROCESS_DB"."AUTO BUFF" <> 195) AND ("MFG PROCESS_DB"."MATERIAL SUCTION"."MATERIAL SUCTION BUFF" <> 5) AND ("MFG PROCESS_DB"."MATERIAL SUCTION"."MATERIAL SUCTION BUFF" <> 10) THEN
       "HYST AND TEMP CUTOFF  DB"."AUTO MOVE PV"."MFG_LOAD CELL" := "AI SCALING DB".PV."SYRUP LOAD CELL";
   END_IF;
END_REGION

REGION Network 15: AUTO SUB HYSTERISIS
   RUNG wire#powerrail
      Contact( "AlwaysTRUE" )
      wire#w1
      Add(in1 := "HYST AND TEMP CUTOFF  DB"."AUTO MOVE PV"."MFG_LOAD CELL", in2 := "HYST AND TEMP CUTOFF  DB"."AUTO MAIN SET PARAMETER"."MFG LOAD CELL", out => "HYST AND TEMP CUTOFF  DB"."AUTO NEW VALUE"."MFG LOAD CELL")
   END_RUNG
   RUNG wire#w1
      "@LOAD CALCULATE"("MFG PROCESS BUFF" := "MFG PROCESS_DB"."AUTO BUFF", "MATERIAL SUCTION BUFF" := "MFG PROCESS_DB"."MATERIAL SUCTION"."MATERIAL SUCTION BUFF", "MOVE PV" := "HYST AND TEMP CUTOFF  DB"."AUTO MOVE PV"."MFG_LOAD CELL", PV := "AI SCALING DB".PV."SYRUP LOAD CELL", "PURIFIED CALCULATE PV" => "MFG PROCESS_DB"."PV PARAMETER"."PURIFIED LOAD", "MATERIAL SORBITOL CALCULATE PV" => "MFG PROCESS_DB"."PV PARAMETER"."MATERIAL_SORBITOL LOAD CELL", "MATERIAL GLUCOSE CALCULATE PV" => "MFG PROCESS_DB"."PV PARAMETER"."MATERIAL_GLUCOSE LOAD CELL", "MATERIAL SUCTION CALCULATE PV" => "MFG PROCESS_DB"."PV PARAMETER"."MATERIAL SUCTION LOAD CELL")
   END_RUNG
   // the same network as SCL:
   IF "AlwaysTRUE" THEN
       "HYST AND TEMP CUTOFF  DB"."AUTO NEW VALUE"."MFG LOAD CELL" := "HYST AND TEMP CUTOFF  DB"."AUTO MOVE PV"."MFG_LOAD CELL" + "HYST AND TEMP CUTOFF  DB"."AUTO MAIN SET PARAMETER"."MFG LOAD CELL";
       "@LOAD CALCULATE"("MFG PROCESS BUFF" := "MFG PROCESS_DB"."AUTO BUFF",
                         "MATERIAL SUCTION BUFF" := "MFG PROCESS_DB"."MATERIAL SUCTION"."MATERIAL SUCTION BUFF",
                         "MOVE PV" := "HYST AND TEMP CUTOFF  DB"."AUTO MOVE PV"."MFG_LOAD CELL",
                         PV := "AI SCALING DB".PV."SYRUP LOAD CELL",
                         "PURIFIED CALCULATE PV" => "MFG PROCESS_DB"."PV PARAMETER"."PURIFIED LOAD",
                         "MATERIAL SORBITOL CALCULATE PV" => "MFG PROCESS_DB"."PV PARAMETER"."MATERIAL_SORBITOL LOAD CELL",
                         "MATERIAL GLUCOSE CALCULATE PV" => "MFG PROCESS_DB"."PV PARAMETER"."MATERIAL_GLUCOSE LOAD CELL",
                         "MATERIAL SUCTION CALCULATE PV" => "MFG PROCESS_DB"."PV PARAMETER"."MATERIAL SUCTION LOAD CELL");
   END_IF;
END_REGION

REGION Network 16: AUTO LOAD CELL CUT OFF
   RUNG wire#powerrail
      Contact( "AlwaysTRUE" )
      wire#w1
      { S7_Templates := "SrcType := Real" } GE_Contact(in1 := "AI SCALING DB".PV."SYRUP LOAD CELL", in2 := "HYST AND TEMP CUTOFF  DB"."AUTO NEW VALUE"."MFG LOAD CELL")
      Move(in := 1, out1 => "LEVEL BUFF".AUTO."MFG LOAD CELL")
   END_RUNG
   RUNG wire#w1
      { S7_Templates := "SrcType := Real" } LT_Contact(in1 := "AI SCALING DB".PV."SYRUP LOAD CELL", in2 := "HYST AND TEMP CUTOFF  DB"."AUTO NEW VALUE"."MFG LOAD CELL")
      Move(in := 0, out1 => "LEVEL BUFF".AUTO."MFG LOAD CELL")
   END_RUNG
   // the same network as SCL:
   IF "AlwaysTRUE" AND ("AI SCALING DB".PV."SYRUP LOAD CELL" >= "HYST AND TEMP CUTOFF  DB"."AUTO NEW VALUE"."MFG LOAD CELL") THEN
       "LEVEL BUFF".AUTO."MFG LOAD CELL" := 1;
   END_IF;
   IF "AlwaysTRUE" AND ("AI SCALING DB".PV."SYRUP LOAD CELL" < "HYST AND TEMP CUTOFF  DB"."AUTO NEW VALUE"."MFG LOAD CELL") THEN
       "LEVEL BUFF".AUTO."MFG LOAD CELL" := 0;
   END_IF;
END_REGION

REGION Network 17: AUTO MFG TEMP MIN_MAX BUFF
